LIN {X 0.201,Y -554.749,Z 1469.573,A 0.000,B 0.000,C 90.000,E1 139.013} C_DIS
LIN {X -0.001,Y -555.947,Z 1469.566,A 0.000,B 0.000,C 90.000,E1 137.919} C_DIS
LIN {X -0.117,Y -557.300,Z 1469.559,A 0.000,B 0.000,C 90.000,E1 136.539} C_DIS
LIN {X 0.103,Y -558.249,Z 1469.552,A 0.000,B 0.000,C 90.000,E1 135.405} C_DIS
LIN {X 0.340,Y -559.051,Z 1469.546,A 0.000,B 0.000,C 90.000,E1 134.271} C_DIS
LIN {X 0.127,Y -559.624,Z 1469.542,A 0.000,B 0.000,C 90.000,E1 133.461} C_DIS
LIN {X 0.073,Y -560.260,Z 1469.534,A 0.000,B 0.000,C 90.000,E1 132.081} C_DIS
LIN {X -0.054,Y -560.649,Z 1469.528,A 0.000,B 0.000,C 90.000,E1 130.987} C_DIS
LIN {X -0.119,Y -560.823,Z 1469.522,A 0.000,B 0.000,C 90.000,E1 129.886} C_DIS
LIN {X -0.071,Y -560.958,Z 1469.512,A 0.000,B 0.000,C 90.000,E1 128.222} C_DIS
LIN {X -0.281,Y -561.117,Z 1469.503,A 0.000,B 0.000,C 90.000,E1 126.583} C_DIS
LIN {X 0.009,Y -561.144,Z 1469.499,A 0.000,B 0.000,C 90.000,E1 125.724} C_DIS
LIN {X 0.070,Y -560.901,Z 1469.492,A 0.000,B 0.000,C 90.000,E1 124.612} C_DIS
LIN {X -0.171,Y -560.446,Z 1469.475,A 0.000,B 0.000,C 90.000,E1 121.592} C_DIS
LIN {X 0.273,Y -560.571,Z 1469.463,A 0.000,B 0.000,C 90.000,E1 119.333} C_DIS
LIN {X -0.178,Y -560.837,Z 1469.454,A 0.000,B 0.000,C 90.000,E1 117.719} C_DIS
LIN {X -0.115,Y -561.178,Z 1469.445,A 0.000,B 0.000,C 90.000,E1 116.052} C_DIS
LIN {X 0.259,Y -561.729,Z 1469.434,A 0.000,B 0.000,C 90.000,E1 114.079} C_DIS
LIN {X 0.068,Y -562.198,Z 1469.426,A 0.000,B 0.000,C 90.000,E1 112.717} C_DIS
LIN {X 0.210,Y -562.729,Z 1469.417,A 0.000,B 0.000,C 90.000,E1 111.046} C_DIS
LIN {X -0.057,Y -563.216,Z 1469.406,A 0.000,B 0.000,C 90.000,E1 109.141} C_DIS
LIN {X -0.074,Y -563.557,Z 1469.399,A 0.000,B 0.000,C 90.000,E1 107.764} C_DIS
LIN {X -0.154,Y -564.110,Z 1469.388,A 0.000,B 0.000,C 90.000,E1 105.843} C_DIS
LIN {X 0.159,Y -564.750,Z 1469.377,A 0.000,B 0.000,C 90.000,E1 103.883} C_DIS
LIN {X -0.160,Y -565.614,Z 1469.365,A 0.000,B 0.000,C 90.000,E1 101.715} C_DIS
LIN {X -0.004,Y -566.581,Z 1469.353,A 0.000,B 0.000,C 90.000,E1 99.500} C_DIS
LIN {X -0.090,Y -567.411,Z 1469.342,A 0.000,B 0.000,C 90.000,E1 97.587} C_DIS
LIN {X -0.232,Y -568.473,Z 1469.332,A 0.000,B 0.000,C 90.000,E1 95.682} C_DIS
LIN {X -0.289,Y -569.933,Z 1469.319,A 0.000,B 0.000,C 90.000,E1 93.498} C_DIS
LIN {X 0.091,Y -571.319,Z 1469.309,A 0.000,B 0.000,C 90.000,E1 91.547} C_DIS
LIN {X 0.042,Y -573.033,Z 1469.297,A 0.000,B 0.000,C 90.000,E1 89.370} C_DIS
LIN {X -0.237,Y -574.312,Z 1469.287,A 0.000,B 0.000,C 90.000,E1 87.764} C_DIS
LIN {X 0.267,Y -575.826,Z 1469.277,A 0.000,B 0.000,C 90.000,E1 85.812} C_DIS
LIN {X 0.077,Y -577.153,Z 1469.268,A 0.000,B 0.000,C 90.000,E1 84.204} C_DIS
LIN {X 0.174,Y -578.805,Z 1469.257,A 0.000,B 0.000,C 90.000,E1 82.299} C_DIS
LIN {X -0.181,Y -580.471,Z 1469.247,A 0.000,B 0.000,C 90.000,E1 80.443} C_DIS
LIN {X -0.058,Y -581.907,Z 1469.238,A 0.000,B 0.000,C 90.000,E1 78.814} C_DIS
LIN {X -0.125,Y -583.585,Z 1469.227,A 0.000,B 0.000,C 90.000,E1 76.937} C_DIS
LIN {X 0.019,Y -584.286,Z 1469.223,A 0.000,B 0.000,C 90.000,E1 76.117} C_DIS
LIN {X -0.015,Y -585.019,Z 1469.217,A 0.000,B 0.000,C 90.000,E1 75.046} C_DIS
LIN {X -0.127,Y -585.954,Z 1469.208,A 0.000,B 0.000,C 90.000,E1 73.449} C_DIS
LIN {X 0.114,Y -586.813,Z 1469.199,A 0.000,B 0.000,C 90.000,E1 71.819} C_DIS
LIN {X -0.177,Y -587.738,Z 1469.190,A 0.000,B 0.000,C 90.000,E1 70.242} C_DIS
LIN {X -0.122,Y -588.454,Z 1469.183,A 0.000,B 0.000,C 90.000,E1 68.901} C_DIS
LIN {X 0.129,Y -589.641,Z 1469.171,A 0.000,B 0.000,C 90.000,E1 66.741} C_DIS
LIN {X -0.084,Y -590.787,Z 1469.161,A 0.000,B 0.000,C 90.000,E1 64.897} C_DIS
LIN {X -0.156,Y -591.847,Z 1469.152,A 0.000,B 0.000,C 90.000,E1 63.307} C_DIS
LIN {X -0.334,Y -593.772,Z 1469.137,A 0.000,B 0.000,C 90.000,E1 60.667} C_DIS
LIN {X -0.115,Y -595.362,Z 1469.127,A 0.000,B 0.000,C 90.000,E1 58.791} C_DIS
LIN {X 0.370,Y -597.188,Z 1469.115,A 0.000,B 0.000,C 90.000,E1 56.628} C_DIS
LIN {X 0.022,Y -598.277,Z 1469.108,A 0.000,B 0.000,C 90.000,E1 55.341} C_DIS
LIN {X -0.114,Y -599.280,Z 1469.100,A 0.000,B 0.000,C 90.000,E1 54.036} C_DIS
LIN {X -0.089,Y -600.482,Z 1469.090,A 0.000,B 0.000,C 90.000,E1 52.190} C_DIS
LIN {X -0.177,Y -601.393,Z 1469.083,A 0.000,B 0.000,C 90.000,E1 50.884} C_DIS
LIN {X -0.118,Y -601.869,Z 1469.077,A 0.000,B 0.000,C 90.000,E1 49.828} C_DIS
LIN {X -0.016,Y -602.241,Z 1469.068,A 0.000,B 0.000,C 90.000,E1 48.243} C_DIS
LIN {X 0.047,Y -602.454,Z 1469.062,A 0.000,B 0.000,C 90.000,E1 47.187} C_DIS
LIN {X -0.325,Y -602.466,Z 1469.053,A 0.000,B 0.000,C 90.000,E1 45.648} C_DIS
LIN {X 0.365,Y -601.994,Z 1469.046,A 0.000,B 0.000,C 90.000,E1 44.271} C_DIS
LIN {X -0.249,Y -601.593,Z 1469.042,A 0.000,B 0.000,C 90.000,E1 43.542} C_DIS
LIN {X 0.211,Y -600.855,Z 1469.036,A 0.000,B 0.000,C 90.000,E1 42.447} C_DIS
LIN {X -0.191,Y -599.900,Z 1469.030,A 0.000,B 0.000,C 90.000,E1 41.434} C_DIS
LIN {X -0.157,Y -598.721,Z 1469.024,A 0.000,B 0.000,C 90.000,E1 40.378} C_DIS
LIN {X 0.320,Y -597.355,Z 1469.018,A 0.000,B 0.000,C 90.000,E1 39.277} C_DIS
LIN {X -0.056,Y -595.749,Z 1469.013,A 0.000,B 0.000,C 90.000,E1 38.257} C_DIS
LIN {X 0.157,Y -594.560,Z 1469.008,A 0.000,B 0.000,C 90.000,E1 37.443} C_DIS
LIN {X -0.047,Y -592.134,Z 1469.001,A 0.000,B 0.000,C 90.000,E1 36.137} C_DIS
LIN {X -0.163,Y -589.103,Z 1468.993,A 0.000,B 0.000,C 90.000,E1 34.818} C_DIS
LIN {X 0.295,Y -586.164,Z 1468.987,A 0.000,B 0.000,C 90.000,E1 33.706} C_DIS
LIN {X -0.280,Y -583.793,Z 1468.983,A 0.000,B 0.000,C 90.000,E1 32.959} C_DIS
LIN {X -0.073,Y -581.068,Z 1468.979,A 0.000,B 0.000,C 90.000,E1 32.133} C_DIS
LIN {X -0.203,Y -578.020,Z 1468.974,A 0.000,B 0.000,C 90.000,E1 31.337} C_DIS
LIN {X -0.066,Y -574.598,Z 1468.969,A 0.000,B 0.000,C 90.000,E1 30.512} C_DIS
LIN {X 0.312,Y -571.404,Z 1468.966,A 0.000,B 0.000,C 90.000,E1 29.795} C_DIS
LIN {X 0.075,Y -567.170,Z 1468.961,A 0.000,B 0.000,C 90.000,E1 28.999} C_DIS
LIN {X -0.288,Y -564.172,Z 1468.958,A 0.000,B 0.000,C 90.000,E1 28.487} C_DIS
LIN {X -0.003,Y -560.134,Z 1468.954,A 0.000,B 0.000,C 90.000,E1 27.769} C_DIS
LIN {X -0.016,Y -555.858,Z 1468.950,A 0.000,B 0.000,C 90.000,E1 27.078} C_DIS
LIN {X -0.155,Y -548.245,Z 1468.944,A 0.000,B 0.000,C 90.000,E1 25.976} C_DIS
LIN {X 0.206,Y -540.958,Z 1468.939,A 0.000,B 0.000,C 90.000,E1 24.951} C_DIS
LIN {X 0.029,Y -535.255,Z 1468.935,A 0.000,B 0.000,C 90.000,E1 24.259} C_DIS
LIN {X 0.142,Y -528.093,Z 1468.930,A 0.000,B 0.000,C 90.000,E1 23.387} C_DIS
LIN {X 0.221,Y -523.920,Z 1468.928,A 0.000,B 0.000,C 90.000,E1 22.950} C_DIS
LIN {X -0.100,Y -520.939,Z 1468.926,A 0.000,B 0.000,C 90.000,E1 22.717} C_DIS
LIN {X -0.056,Y -517.716,Z 1468.925,A 0.000,B 0.000,C 90.000,E1 22.461} C_DIS
LIN {X 0.056,Y -516.052,Z 1468.924,A 0.000,B 0.000,C 90.000,E1 22.333} C_DIS
LIN {X 0.011,Y -512.686,Z 1468.923,A 0.000,B 0.000,C 90.000,E1 22.153} C_DIS
LIN {X 0.005,Y -510.601,Z 1468.923,A 0.000,B 0.000,C 90.000,E1 22.078} C_DIS
LIN {X -0.187,Y -509.425,Z 1468.923,A 0.000,B 0.000,C 90.000,E1 22.078} C_DIS
LIN {X 0.188,Y -378.596,Z 1468.923,A 0.000,B 0.000,C 90.000,E1 22.025} C_DIS
LIN {X 0.122,Y -373.766,Z 1468.898,A 0.000,B 0.000,C 90.000,E1 17.638} C_DIS
LIN {X 0.069,Y -372.871,Z 1468.894,A 0.000,B 0.000,C 90.000,E1 16.913} C_DIS
LIN {X -0.029,Y -367.601,Z 1468.865,A 0.000,B 0.000,C 90.000,E1 11.771} C_DIS
LIN {X 0.055,Y -366.481,Z 1468.855,A 0.000,B 0.000,C 90.000,E1 9.905} C_DIS
LIN {X -0.009,Y -361.784,Z 1468.822,A 0.000,B 0.000,C 90.000,E1 3.955} C_DIS
LIN {X -0.123,Y -360.899,Z 1468.801,A 0.000,B 0.000,C 90.000,E1 0.229} C_DIS
LIN {X -0.053,Y -359.426,Z 1468.770,A 0.000,B 0.000,C 90.000,E1 354.546} C_DIS
LIN {X 0.070,Y -358.890,Z 1468.759,A 0.000,B 0.000,C 90.000,E1 352.648} C_DIS
LIN {X -0.020,Y -359.563,Z 1468.726,A 0.000,B 0.000,C 90.000,E1 346.645} C_DIS
LIN {X 0.001,Y -361.801,Z 1468.684,A 0.000,B 0.000,C 90.000,E1 339.135} C_DIS
LIN {X -0.154,Y -362.053,Z 1468.680,A 0.000,B 0.000,C 90.000,E1 338.411} C_DIS
LIN {X 0.189,Y -365.980,Z 1468.643,A 0.000,B 0.000,C 90.000,E1 331.641} C_DIS
LIN {X 0.029,Y -366.387,Z 1468.639,A 0.000,B 0.000,C 90.000,E1 330.923} C_DIS
LIN {X -0.031,Y -371.355,Z 1468.604,A 0.000,B 0.000,C 90.000,E1 324.642} C_DIS
LIN {X -0.043,Y -371.766,Z 1468.602,A 0.000,B 0.000,C 90.000,E1 324.276} C_DIS
LIN {X 0.013,Y -377.358,Z 1468.567,A 0.000,B 0.000,C 90.000,E1 318.038} C_DIS
LIN {X 0.012,Y -378.235,Z 1468.563,A 0.000,B 0.000,C 90.000,E1 317.310} C_DIS
LIN {X 0.002,Y -383.940,Z 1468.531,A 0.000,B 0.000,C 90.000,E1 311.515} C_DIS
LIN {X 0.088,Y -384.893,Z 1468.527,A 0.000,B 0.000,C 90.000,E1 310.782} C_DIS
LIN {X 0.262,Y -390.610,Z 1468.495,A 0.000,B 0.000,C 90.000,E1 305.025} C_DIS
LIN {X 0.106,Y -391.104,Z 1468.493,A 0.000,B 0.000,C 90.000,E1 304.692} C_DIS
LIN {X 0.022,Y -391.648,Z 1468.489,A 0.000,B 0.000,C 90.000,E1 303.992} C_DIS
LIN {X -0.080,Y -396.825,Z 1468.459,A 0.000,B 0.000,C 90.000,E1 298.693} C_DIS
LIN {X -0.210,Y -397.120,Z 1468.457,A 0.000,B 0.000,C 90.000,E1 298.359} C_DIS
LIN {X -0.055,Y -401.597,Z 1468.426,A 0.000,B 0.000,C 90.000,E1 292.717} C_DIS
LIN {X 0.222,Y -404.659,Z 1468.395,A 0.000,B 0.000,C 90.000,E1 287.094} C_DIS
LIN {X -0.079,Y -404.735,Z 1468.391,A 0.000,B 0.000,C 90.000,E1 286.441} C_DIS
LIN {X 0.214,Y -406.099,Z 1468.364,A 0.000,B 0.000,C 90.000,E1 281.535} C_DIS
LIN {X -0.176,Y -406.094,Z 1468.362,A 0.000,B 0.000,C 90.000,E1 281.243} C_DIS
LIN {X -0.097,Y -405.680,Z 1468.333,A 0.000,B 0.000,C 90.000,E1 276.024} C_DIS
LIN {X -0.165,Y -405.058,Z 1468.328,A 0.000,B 0.000,C 90.000,E1 274.992} C_DIS
LIN {X -0.060,Y -403.497,Z 1468.304,A 0.000,B 0.000,C 90.000,E1 270.802} C_DIS
LIN {X -0.092,Y -403.288,Z 1468.302,A 0.000,B 0.000,C 90.000,E1 270.458} C_DIS
LIN {X 0.091,Y -398.931,Z 1468.271,A 0.000,B 0.000,C 90.000,E1 264.837} C_DIS
LIN {X -0.040,Y -393.108,Z 1468.242,A 0.000,B 0.000,C 90.000,E1 259.567} C_DIS
LIN {X -0.079,Y -392.835,Z 1468.240,A 0.000,B 0.000,C 90.000,E1 259.218} C_DIS
LIN {X 0.034,Y -385.993,Z 1468.212,A 0.000,B 0.000,C 90.000,E1 254.212} C_DIS
LIN {X -0.026,Y -385.267,Z 1468.208,A 0.000,B 0.000,C 90.000,E1 253.504} C_DIS
LIN {X -0.004,Y -384.768,Z 1468.206,A 0.000,B 0.000,C 90.000,E1 253.142} C_DIS
LIN {X 0.221,Y -377.973,Z 1468.182,A 0.000,B 0.000,C 90.000,E1 248.773} C_DIS
LIN {X -0.044,Y -376.233,Z 1468.174,A 0.000,B 0.000,C 90.000,E1 247.358} C_DIS
LIN {X 0.057,Y -374.944,Z 1468.170,A 0.000,B 0.000,C 90.000,E1 246.613} C_DIS
LIN {X -0.208,Y -368.417,Z 1468.148,A 0.000,B 0.000,C 90.000,E1 242.615} C_DIS
LIN {X 0.097,Y -366.047,Z 1468.137,A 0.000,B 0.000,C 90.000,E1 240.717} C_DIS
LIN {X 0.004,Y -359.196,Z 1468.115,A 0.000,B 0.000,C 90.000,E1 236.628} C_DIS
LIN {X 0.021,Y -355.842,Z 1468.100,A 0.000,B 0.000,C 90.000,E1 233.989} C_DIS
LIN {X -0.173,Y -348.793,Z 1468.075,A 0.000,B 0.000,C 90.000,E1 229.461} C_DIS
LIN {X -0.097,Y -346.185,Z 1468.062,A 0.000,B 0.000,C 90.000,E1 227.148} C_DIS
LIN {X -0.088,Y -345.065,Z 1468.058,A 0.000,B 0.000,C 90.000,E1 226.377} C_DIS
LIN {X 0.094,Y -338.586,Z 1468.030,A 0.000,B 0.000,C 90.000,E1 221.310} C_DIS
LIN {X 0.094,Y -336.840,Z 1468.019,A 0.000,B 0.000,C 90.000,E1 219.358} C_DIS
LIN {X 0.014,Y -330.861,Z 1467.988,A 0.000,B 0.000,C 90.000,E1 213.865} C_DIS
LIN {X 0.149,Y -329.296,Z 1467.975,A 0.000,B 0.000,C 90.000,E1 211.465} C_DIS
LIN {X -0.154,Y -324.669,Z 1467.942,A 0.000,B 0.000,C 90.000,E1 205.540} C_DIS
LIN {X 0.174,Y -323.837,Z 1467.928,A 0.000,B 0.000,C 90.000,E1 203.078} C_DIS
LIN {X -0.017,Y -321.124,Z 1467.881,A 0.000,B 0.000,C 90.000,E1 194.662} C_DIS
LIN {X 0.138,Y -320.932,Z 1467.877,A 0.000,B 0.000,C 90.000,E1 193.828} C_DIS
LIN {X -0.076,Y -321.562,Z 1467.832,A 0.000,B 0.000,C 90.000,E1 185.796} C_DIS
LIN {X -0.143,Y -324.415,Z 1467.790,A 0.000,B 0.000,C 90.000,E1 178.165} C_DIS
LIN {X -0.141,Y -325.376,Z 1467.783,A 0.000,B 0.000,C 90.000,E1 176.963} C_DIS
LIN {X -0.100,Y -329.112,Z 1467.750,A 0.000,B 0.000,C 90.000,E1 170.971} C_DIS
LIN {X 0.061,Y -334.260,Z 1467.726,A 0.000,B 0.000,C 90.000,E1 166.589} C_DIS
LIN {X 0.067,Y -335.488,Z 1467.719,A 0.000,B 0.000,C 90.000,E1 165.408} C_DIS
LIN {X 0.143,Y -340.932,Z 1467.695,A 0.000,B 0.000,C 90.000,E1 161.094} C_DIS
LIN {X -0.172,Y -342.138,Z 1467.691,A 0.000,B 0.000,C 90.000,E1 160.369} C_DIS
LIN {X 0.102,Y -347.570,Z 1467.668,A 0.000,B 0.000,C 90.000,E1 156.305} C_DIS
LIN {X 0.097,Y -466.149,Z 1467.668,A 0.000,B 0.000,C 90.000,E1 156.305} C_DIS
LIN {X 0.196,Y -469.174,Z 1467.668,A 0.000,B 0.000,C 90.000,E1 156.230} C_DIS
LIN {X -0.079,Y -473.073,Z 1467.667,A 0.000,B 0.000,C 90.000,E1 156.102} C_DIS
LIN {X 0.134,Y -475.940,Z 1467.666,A 0.000,B 0.000,C 90.000,E1 155.921} C_DIS
LIN {X 0.123,Y -478.786,Z 1467.665,A 0.000,B 0.000,C 90.000,E1 155.741} C_DIS
LIN {X 0.219,Y -483.218,Z 1467.664,A 0.000,B 0.000,C 90.000,E1 155.409} C_DIS
LIN {X -0.194,Y -488.987,Z 1467.661,A 0.000,B 0.000,C 90.000,E1 154.973} C_DIS
LIN {X -0.117,Y -497.335,Z 1467.656,A 0.000,B 0.000,C 90.000,E1 154.152} C_DIS
LIN {X 0.163,Y -500.136,Z 1467.655,A 0.000,B 0.000,C 90.000,E1 153.845} C_DIS
LIN {X -0.135,Y -505.377,Z 1467.652,A 0.000,B 0.000,C 90.000,E1 153.307} C_DIS
LIN {X 0.082,Y -510.366,Z 1467.648,A 0.000,B 0.000,C 90.000,E1 152.692} C_DIS
LIN {X 0.062,Y -514.904,Z 1467.645,A 0.000,B 0.000,C 90.000,E1 152.103} C_DIS
LIN {X 0.071,Y -518.945,Z 1467.642,A 0.000,B 0.000,C 90.000,E1 151.513} C_DIS
LIN {X 0.111,Y -522.546,Z 1467.639,A 0.000,B 0.000,C 90.000,E1 150.923} C_DIS
LIN {X 0.179,Y -525.767,Z 1467.635,A 0.000,B 0.000,C 90.000,E1 150.333} C_DIS
LIN {X 0.115,Y -529.332,Z 1467.631,A 0.000,B 0.000,C 90.000,E1 149.616} C_DIS
LIN {X -0.227,Y -531.880,Z 1467.628,A 0.000,B 0.000,C 90.000,E1 149.076} C_DIS
LIN {X 0.181,Y -534.218,Z 1467.625,A 0.000,B 0.000,C 90.000,E1 148.456} C_DIS
LIN {X 0.321,Y -537.331,Z 1467.620,A 0.000,B 0.000,C 90.000,E1 147.582} C_DIS
LIN {X 0.041,Y -540.071,Z 1467.615,A 0.000,B 0.000,C 90.000,E1 146.755} C_DIS
LIN {X 0.240,Y -542.557,Z 1467.611,A 0.000,B 0.000,C 90.000,E1 145.881} C_DIS
LIN {X 0.010,Y -544.834,Z 1467.606,A 0.000,B 0.000,C 90.000,E1 145.055} C_DIS
LIN {X 0.160,Y -547.458,Z 1467.600,A 0.000,B 0.000,C 90.000,E1 143.909} C_DIS
LIN {X 0.022,Y -549.701,Z 1467.593,A 0.000,B 0.000,C 90.000,E1 142.798} C_DIS
LIN {X -0.253,Y -551.173,Z 1467.589,A 0.000,B 0.000,C 90.000,E1 141.984} C_DIS
LIN {X 0.330,Y -552.833,Z 1467.583,A 0.000,B 0.000,C 90.000,E1 140.803} C_DIS
LIN {X 0.159,Y -554.204,Z 1467.576,A 0.000,B 0.000,C 90.000,E1 139.703} C_DIS
LIN {X 0.010,Y -555.758,Z 1467.568,A 0.000,B 0.000,C 90.000,E1 138.324} C_DIS
LIN {X -0.072,Y -557.378,Z 1467.559,A 0.000,B 0.000,C 90.000,E1 136.662} C_DIS
LIN {X -0.235,Y -558.335,Z 1467.553,A 0.000,B 0.000,C 90.000,E1 135.567} C_DIS
LIN {X 0.003,Y -559.169,Z 1467.547,A 0.000,B 0.000,C 90.000,E1 134.433} C_DIS
LIN {X -0.085,Y -559.968,Z 1467.539,A 0.000,B 0.000,C 90.000,E1 133.056} C_DIS
LIN {X -0.136,Y -560.558,Z 1467.531,A 0.000,B 0.000,C 90.000,E1 131.676} C_DIS
LIN {X -0.177,Y -560.849,Z 1467.524,A 0.000,B 0.000,C 90.000,E1 130.297} C_DIS
LIN {X -0.146,Y -560.969,Z 1467.516,A 0.000,B 0.000,C 90.000,E1 128.910} C_DIS
LIN {X 0.091,Y -561.146,Z 1467.505,A 0.000,B 0.000,C 90.000,E1 126.950} C_DIS
LIN {X 0.027,Y -561.184,Z 1467.499,A 0.000,B 0.000,C 90.000,E1 125.851} C_DIS
LIN {X -0.012,Y -561.036,Z 1467.495,A 0.000,B 0.000,C 90.000,E1 125.025} C_DIS
LIN {X -0.033,Y -560.452,Z 1467.479,A 0.000,B 0.000,C 90.000,E1 122.260} C_DIS
LIN {X -0.151,Y -560.474,Z 1467.469,A 0.000,B 0.000,C 90.000,E1 120.335} C_DIS
LIN {X 0.024,Y -560.750,Z 1467.456,A 0.000,B 0.000,C 90.000,E1 118.103} C_DIS
LIN {X 0.082,Y -561.087,Z 1467.447,A 0.000,B 0.000,C 90.000,E1 116.437} C_DIS
LIN {X 0.259,Y -561.706,Z 1467.435,A 0.000,B 0.000,C 90.000,E1 114.207} C_DIS
LIN {X -0.132,Y -562.266,Z 1467.425,A 0.000,B 0.000,C 90.000,E1 112.589} C_DIS
LIN {X 0.008,Y -562.769,Z 1467.416,A 0.000,B 0.000,C 90.000,E1 110.918} C_DIS
LIN {X 0.270,Y -563.294,Z 1467.406,A 0.000,B 0.000,C 90.000,E1 108.960} C_DIS
LIN {X -0.205,Y -563.516,Z 1467.401,A 0.000,B 0.000,C 90.000,E1 108.181} C_DIS
LIN {X -0.289,Y -564.022,Z 1467.390,A 0.000,B 0.000,C 90.000,E1 106.260} C_DIS
LIN {X 0.187,Y -564.730,Z 1467.378,A 0.000,B 0.000,C 90.000,E1 104.008} C_DIS
LIN {X -0.005,Y -565.596,Z 1467.366,A 0.000,B 0.000,C 90.000,E1 101.827} C_DIS
LIN {X -0.029,Y -566.416,Z 1467.355,A 0.000,B 0.000,C 90.000,E1 99.905} C_DIS
LIN {X 0.181,Y -567.017,Z 1467.347,A 0.000,B 0.000,C 90.000,E1 98.511} C_DIS
LIN {X -0.264,Y -568.258,Z 1467.334,A 0.000,B 0.000,C 90.000,E1 96.087} C_DIS
LIN {X -0.159,Y -569.888,Z 1467.320,A 0.000,B 0.000,C 90.000,E1 93.612} C_DIS
LIN {X 0.220,Y -571.259,Z 1467.309,A 0.000,B 0.000,C 90.000,E1 91.661} C_DIS
LIN {X -0.111,Y -572.525,Z 1467.300,A 0.000,B 0.000,C 90.000,E1 90.057} C_DIS
LIN {X 0.018,Y -573.646,Z 1467.293,A 0.000,B 0.000,C 90.000,E1 88.682} C_DIS
LIN {X -0.252,Y -574.959,Z 1467.284,A 0.000,B 0.000,C 90.000,E1 87.078} C_DIS
LIN {X 0.110,Y -576.250,Z 1467.275,A 0.000,B 0.000,C 90.000,E1 85.412} C_DIS
LIN {X -0.224,Y -577.403,Z 1467.267,A 0.000,B 0.000,C 90.000,E1 84.090} C_DIS
LIN {X -0.125,Y -579.057,Z 1467.257,A 0.000,B 0.000,C 90.000,E1 82.186} C_DIS
LIN {X 0.092,Y -580.736,Z 1467.246,A 0.000,B 0.000,C 90.000,E1 80.274} C_DIS
LIN {X 0.327,Y -582.230,Z 1467.237,A 0.000,B 0.000,C 90.000,E1 78.634} C_DIS
LIN {X -0.053,Y -584.147,Z 1467.225,A 0.000,B 0.000,C 90.000,E1 76.520} C_DIS
LIN {X 0.098,Y -584.759,Z 1467.221,A 0.000,B 0.000,C 90.000,E1 75.700} C_DIS
LIN {X 0.073,Y -585.441,Z 1467.215,A 0.000,B 0.000,C 90.000,E1 74.629} C_DIS
LIN {X 0.138,Y -586.351,Z 1467.206,A 0.000,B 0.000,C 90.000,E1 73.015} C_DIS
LIN {X 0.214,Y -587.207,Z 1467.197,A 0.000,B 0.000,C 90.000,E1 71.402} C_DIS
LIN {X 0.258,Y -588.014,Z 1467.189,A 0.000,B 0.000,C 90.000,E1 70.061} C_DIS
LIN {X 0.194,Y -588.824,Z 1467.181,A 0.000,B 0.000,C 90.000,E1 68.465} C_DIS
LIN {X 0.141,Y -589.732,Z 1467.172,A 0.000,B 0.000,C 90.000,E1 66.869} C_DIS
LIN {X -0.074,Y -590.881,Z 1467.161,A 0.000,B 0.000,C 90.000,E1 65.025} C_DIS
LIN {X 0.284,Y -592.149,Z 1467.151,A 0.000,B 0.000,C 90.000,E1 63.127} C_DIS
LIN {X -0.121,Y -594.089,Z 1467.136,A 0.000,B 0.000,C 90.000,E1 60.511} C_DIS
LIN {X -0.189,Y -595.677,Z 1467.126,A 0.000,B 0.000,C 90.000,E1 58.663} C_DIS
LIN {X 0.074,Y -597.286,Z 1467.116,A 0.000,B 0.000,C 90.000,E1 56.786} C_DIS
LIN {X 0.295,Y -598.634,Z 1467.107,A 0.000,B 0.000,C 90.000,E1 55.182} C_DIS
LIN {X -0.182,Y -599.616,Z 1467.099,A 0.000,B 0.000,C 90.000,E1 53.909} C_DIS
LIN {X -0.157,Y -600.796,Z 1467.089,A 0.000,B 0.000,C 90.000,E1 52.065} C_DIS
LIN {X -0.113,Y -601.577,Z 1467.083,A 0.000,B 0.000,C 90.000,E1 51.009} C_DIS
LIN {X -0.046,Y -602.091,Z 1467.078,A 0.000,B 0.000,C 90.000,E1 49.952} C_DIS
LIN {X 0.313,Y -602.538,Z 1467.067,A 0.000,B 0.000,C 90.000,E1 48.081} C_DIS
LIN {X -0.061,Y -602.725,Z 1467.062,A 0.000,B 0.000,C 90.000,E1 47.067} C_DIS
LIN {X 0.217,Y -602.743,Z 1467.054,A 0.000,B 0.000,C 90.000,E1 45.729} C_DIS
LIN {X 0.039,Y -602.531,Z 1467.050,A 0.000,B 0.000,C 90.000,E1 44.960} C_DIS
LIN {X 0.302,Y -601.979,Z 1467.043,A 0.000,B 0.000,C 90.000,E1 43.623} C_DIS
LIN {X 0.125,Y -601.440,Z 1467.038,A 0.000,B 0.000,C 90.000,E1 42.852} C_DIS
LIN {X -0.028,Y -600.376,Z 1467.031,A 0.000,B 0.000,C 90.000,E1 41.553} C_DIS
LIN {X -0.198,Y -598.867,Z 1467.024,A 0.000,B 0.000,C 90.000,E1 40.253} C_DIS
LIN {X -0.175,Y -597.455,Z 1467.018,A 0.000,B 0.000,C 90.000,E1 39.197} C_DIS
LIN {X -0.092,Y -595.069,Z 1467.009,A 0.000,B 0.000,C 90.000,E1 37.604} C_DIS
LIN {X -0.113,Y -594.169,Z 1467.006,A 0.000,B 0.000,C 90.000,E1 37.076} C_DIS
LIN {X -0.061,Y -592.208,Z 1467.000,A 0.000,B 0.000,C 90.000,E1 36.011} C_DIS
LIN {X -0.172,Y -589.101,Z 1466.993,A 0.000,B 0.000,C 90.000,E1 34.692} C_DIS
LIN {X -0.333,Y -585.389,Z 1466.985,A 0.000,B 0.000,C 90.000,E1 33.372} C_DIS
LIN {X 0.033,Y -583.794,Z 1466.982,A 0.000,B 0.000,C 90.000,E1 32.801} C_DIS
LIN {X -0.074,Y -581.018,Z 1466.978,A 0.000,B 0.000,C 90.000,E1 32.005} C_DIS
LIN {X -0.202,Y -577.937,Z 1466.973,A 0.000,B 0.000,C 90.000,E1 31.209} C_DIS
LIN {X -0.066,Y -574.532,Z 1466.969,A 0.000,B 0.000,C 90.000,E1 30.384} C_DIS
LIN {X 0.312,Y -571.272,Z 1466.965,A 0.000,B 0.000,C 90.000,E1 29.667} C_DIS
LIN {X 0.075,Y -567.034,Z 1466.960,A 0.000,B 0.000,C 90.000,E1 28.871} C_DIS
LIN {X 0.286,Y -562.409,Z 1466.956,A 0.000,B 0.000,C 90.000,E1 28.025} C_DIS
LIN {X 0.086,Y -556.524,Z 1466.951,A 0.000,B 0.000,C 90.000,E1 27.078} C_DIS
LIN {X -0.046,Y -548.994,Z 1466.944,A 0.000,B 0.000,C 90.000,E1 25.976} C_DIS
LIN {X -0.033,Y -540.645,Z 1466.938,A 0.000,B 0.000,C 90.000,E1 24.847} C_DIS
LIN {X 0.153,Y -536.107,Z 1466.935,A 0.000,B 0.000,C 90.000,E1 24.259} C_DIS
LIN {X 0.123,Y -527.736,Z 1466.929,A 0.000,B 0.000,C 90.000,E1 23.259} C_DIS
LIN {X 0.004,Y -522.522,Z 1466.926,A 0.000,B 0.000,C 90.000,E1 22.695} C_DIS
LIN {X 0.003,Y -518.208,Z 1466.924,A 0.000,B 0.000,C 90.000,E1 22.280} C_DIS
LIN {X -0.007,Y -513.505,Z 1466.922,A 0.000,B 0.000,C 90.000,E1 21.897} C_DIS
LIN {X 0.047,Y -511.740,Z 1466.921,A 0.000,B 0.000,C 90.000,E1 21.770} C_DIS
LIN {X 0.031,Y -509.876,Z 1466.920,A 0.000,B 0.000,C 90.000,E1 21.663} C_DIS
LIN {X -0.001,Y -506.943,Z 1466.920,A 0.000,B 0.000,C 90.000,E1 21.535} C_DIS
LIN {X 0.199,Y -504.735,Z 1466.919,A 0.000,B 0.000,C 90.000,E1 21.461} C_DIS
LIN {X 0.124,Y -377.830,Z 1466.919,A 0.000,B 0.000,C 90.000,E1 21.461} C_DIS
LIN {X -0.114,Y -373.501,Z 1466.897,A 0.000,B 0.000,C 90.000,E1 17.402} C_DIS
LIN {X -0.075,Y -367.945,Z 1466.868,A 0.000,B 0.000,C 90.000,E1 12.243} C_DIS
LIN {X -0.056,Y -366.530,Z 1466.856,A 0.000,B 0.000,C 90.000,E1 10.018} C_DIS
LIN {X 0.087,Y -365.038,Z 1466.847,A 0.000,B 0.000,C 90.000,E1 8.511} C_DIS
LIN {X 0.182,Y -361.084,Z 1466.810,A 0.000,B 0.000,C 90.000,E1 1.776} C_DIS
LIN {X 0.123,Y -360.905,Z 1466.802,A 0.000,B 0.000,C 90.000,E1 0.286} C_DIS
LIN {X -0.053,Y -359.426,Z 1466.770,A 0.000,B 0.000,C 90.000,E1 354.546} C_DIS
LIN {X 0.070,Y -358.890,Z 1466.759,A 0.000,B 0.000,C 90.000,E1 352.648} C_DIS
LIN {X -0.020,Y -359.563,Z 1466.726,A 0.000,B 0.000,C 90.000,E1 346.645} C_DIS
LIN {X 0.001,Y -361.801,Z 1466.684,A 0.000,B 0.000,C 90.000,E1 339.135} C_DIS
LIN {X -0.154,Y -362.053,Z 1466.680,A 0.000,B 0.000,C 90.000,E1 338.411} C_DIS
LIN {X 0.189,Y -365.980,Z 1466.643,A 0.000,B 0.000,C 90.000,E1 331.641} C_DIS
LIN {X 0.029,Y -366.387,Z 1466.639,A 0.000,B 0.000,C 90.000,E1 330.923} C_DIS
LIN {X -0.031,Y -371.355,Z 1466.604,A 0.000,B 0.000,C 90.000,E1 324.642} C_DIS
LIN {X -0.043,Y -371.766,Z 1466.602,A 0.000,B 0.000,C 90.000,E1 324.276} C_DIS
LIN {X 0.013,Y -377.358,Z 1466.567,A 0.000,B 0.000,C 90.000,E1 318.038} C_DIS
LIN {X 0.012,Y -378.235,Z 1466.563,A 0.000,B 0.000,C 90.000,E1 317.310} C_DIS
LIN {X 0.002,Y -383.940,Z 1466.531,A 0.000,B 0.000,C 90.000,E1 311.515} C_DIS
LIN {X 0.088,Y -384.893,Z 1466.527,A 0.000,B 0.000,C 90.000,E1 310.782} C_DIS
LIN {X 0.262,Y -390.610,Z 1466.495,A 0.000,B 0.000,C 90.000,E1 305.025} C_DIS
LIN {X 0.106,Y -391.104,Z 1466.493,A 0.000,B 0.000,C 90.000,E1 304.692} C_DIS
LIN {X 0.022,Y -391.648,Z 1466.489,A 0.000,B 0.000,C 90.000,E1 303.992} C_DIS
LIN {X -0.080,Y -396.825,Z 1466.459,A 0.000,B 0.000,C 90.000,E1 298.693} C_DIS
LIN {X -0.210,Y -397.120,Z 1466.457,A 0.000,B 0.000,C 90.000,E1 298.359} C_DIS
LIN {X -0.055,Y -401.597,Z 1466.426,A 0.000,B 0.000,C 90.000,E1 292.717} C_DIS
LIN {X 0.222,Y -404.659,Z 1466.395,A 0.000,B 0.000,C 90.000,E1 287.094} C_DIS
LIN {X -0.079,Y -404.735,Z 1466.391,A 0.000,B 0.000,C 90.000,E1 286.441} C_DIS
LIN {X 0.214,Y -406.099,Z 1466.364,A 0.000,B 0.000,C 90.000,E1 281.535} C_DIS
LIN {X -0.176,Y -406.094,Z 1466.362,A 0.000,B 0.000,C 90.000,E1 281.243} C_DIS
LIN {X -0.097,Y -405.680,Z 1466.333,A 0.000,B 0.000,C 90.000,E1 276.024} C_DIS
LIN {X -0.165,Y -405.058,Z 1466.328,A 0.000,B 0.000,C 90.000,E1 274.992} C_DIS
LIN {X -0.060,Y -403.497,Z 1466.304,A 0.000,B 0.000,C 90.000,E1 270.802} C_DIS
LIN {X -0.092,Y -403.288,Z 1466.302,A 0.000,B 0.000,C 90.000,E1 270.458} C_DIS
LIN {X 0.091,Y -398.931,Z 1466.271,A 0.000,B 0.000,C 90.000,E1 264.837} C_DIS
LIN {X -0.040,Y -393.108,Z 1466.242,A 0.000,B 0.000,C 90.000,E1 259.567} C_DIS
LIN {X -0.079,Y -392.835,Z 1466.240,A 0.000,B 0.000,C 90.000,E1 259.218} C_DIS
LIN {X 0.034,Y -385.993,Z 1466.212,A 0.000,B 0.000,C 90.000,E1 254.212} C_DIS
LIN {X -0.026,Y -385.267,Z 1466.208,A 0.000,B 0.000,C 90.000,E1 253.504} C_DIS
LIN {X -0.004,Y -384.768,Z 1466.206,A 0.000,B 0.000,C 90.000,E1 253.142} C_DIS
LIN {X 0.221,Y -377.973,Z 1466.182,A 0.000,B 0.000,C 90.000,E1 248.773} C_DIS
LIN {X -0.044,Y -376.233,Z 1466.174,A 0.000,B 0.000,C 90.000,E1 247.358} C_DIS
LIN {X 0.057,Y -374.944,Z 1466.170,A 0.000,B 0.000,C 90.000,E1 246.613} C_DIS
LIN {X -0.208,Y -368.417,Z 1466.148,A 0.000,B 0.000,C 90.000,E1 242.615} C_DIS
LIN {X 0.097,Y -366.047,Z 1466.137,A 0.000,B 0.000,C 90.000,E1 240.717} C_DIS
LIN {X 0.004,Y -359.196,Z 1466.115,A 0.000,B 0.000,C 90.000,E1 236.628} C_DIS
LIN {X 0.021,Y -355.842,Z 1466.100,A 0.000,B 0.000,C 90.000,E1 233.989} C_DIS
LIN {X -0.173,Y -348.793,Z 1466.075,A 0.000,B 0.000,C 90.000,E1 229.461} C_DIS
LIN {X -0.097,Y -346.185,Z 1466.062,A 0.000,B 0.000,C 90.000,E1 227.148} C_DIS
LIN {X -0.088,Y -345.065,Z 1466.058,A 0.000,B 0.000,C 90.000,E1 226.377} C_DIS
LIN {X 0.094,Y -338.586,Z 1466.030,A 0.000,B 0.000,C 90.000,E1 221.310} C_DIS
LIN {X 0.094,Y -336.840,Z 1466.019,A 0.000,B 0.000,C 90.000,E1 219.358} C_DIS
LIN {X 0.014,Y -330.861,Z 1465.988,A 0.000,B 0.000,C 90.000,E1 213.865} C_DIS
LIN {X 0.149,Y -329.296,Z 1465.975,A 0.000,B 0.000,C 90.000,E1 211.465} C_DIS
LIN {X -0.154,Y -324.669,Z 1465.942,A 0.000,B 0.000,C 90.000,E1 205.540} C_DIS
LIN {X 0.174,Y -323.837,Z 1465.928,A 0.000,B 0.000,C 90.000,E1 203.078} C_DIS
LIN {X -0.017,Y -321.124,Z 1465.881,A 0.000,B 0.000,C 90.000,E1 194.662} C_DIS
LIN {X 0.138,Y -320.932,Z 1465.877,A 0.000,B 0.000,C 90.000,E1 193.828} C_DIS
LIN {X -0.076,Y -321.562,Z 1465.832,A 0.000,B 0.000,C 90.000,E1 185.796} C_DIS
LIN {X -0.143,Y -324.415,Z 1465.790,A 0.000,B 0.000,C 90.000,E1 178.165} C_DIS
LIN {X -0.141,Y -325.376,Z 1465.783,A 0.000,B 0.000,C 90.000,E1 176.963} C_DIS
LIN {X -0.100,Y -329.112,Z 1465.750,A 0.000,B 0.000,C 90.000,E1 170.971} C_DIS
LIN {X 0.061,Y -334.260,Z 1465.726,A 0.000,B 0.000,C 90.000,E1 166.589} C_DIS
LIN {X 0.067,Y -335.488,Z 1465.719,A 0.000,B 0.000,C 90.000,E1 165.408} C_DIS
LIN {X 0.143,Y -340.932,Z 1465.695,A 0.000,B 0.000,C 90.000,E1 161.094} C_DIS
LIN {X -0.172,Y -342.138,Z 1465.691,A 0.000,B 0.000,C 90.000,E1 160.369} C_DIS
LIN {X 0.043,Y -346.707,Z 1465.672,A 0.000,B 0.000,C 90.000,E1 156.869} C_DIS
LIN {X 0.018,Y -460.252,Z 1465.672,A 0.000,B 0.000,C 90.000,E1 156.869} C_DIS
LIN {X 0.126,Y -463.257,Z 1465.671,A 0.000,B 0.000,C 90.000,E1 156.794} C_DIS
LIN {X -0.145,Y -465.604,Z 1465.671,A 0.000,B 0.000,C 90.000,E1 156.741} C_DIS
LIN {X -0.158,Y -468.354,Z 1465.670,A 0.000,B 0.000,C 90.000,E1 156.613} C_DIS
LIN {X -0.010,Y -471.281,Z 1465.669,A 0.000,B 0.000,C 90.000,E1 156.433} C_DIS
LIN {X 0.134,Y -474.187,Z 1465.668,A 0.000,B 0.000,C 90.000,E1 156.230} C_DIS
LIN {X 0.024,Y -478.628,Z 1465.666,A 0.000,B 0.000,C 90.000,E1 155.921} C_DIS
LIN {X 0.209,Y -484.407,Z 1465.664,A 0.000,B 0.000,C 90.000,E1 155.409} C_DIS
LIN {X -0.158,Y -491.532,Z 1465.660,A 0.000,B 0.000,C 90.000,E1 154.793} C_DIS
LIN {X 0.116,Y -498.552,Z 1465.656,A 0.000,B 0.000,C 90.000,E1 154.076} C_DIS
LIN {X 0.278,Y -502.524,Z 1465.654,A 0.000,B 0.000,C 90.000,E1 153.640} C_DIS
LIN {X -0.164,Y -506.438,Z 1465.651,A 0.000,B 0.000,C 90.000,E1 153.256} C_DIS
LIN {X -0.001,Y -510.230,Z 1465.649,A 0.000,B 0.000,C 90.000,E1 152.794} C_DIS
LIN {X -0.265,Y -514.804,Z 1465.646,A 0.000,B 0.000,C 90.000,E1 152.231} C_DIS
LIN {X -0.258,Y -518.895,Z 1465.642,A 0.000,B 0.000,C 90.000,E1 151.641} C_DIS
LIN {X -0.220,Y -522.519,Z 1465.639,A 0.000,B 0.000,C 90.000,E1 151.051} C_DIS
LIN {X -0.312,Y -526.527,Z 1465.635,A 0.000,B 0.000,C 90.000,E1 150.333} C_DIS
LIN {X -0.105,Y -530.012,Z 1465.631,A 0.000,B 0.000,C 90.000,E1 149.587} C_DIS
LIN {X 0.018,Y -532.561,Z 1465.628,A 0.000,B 0.000,C 90.000,E1 148.997} C_DIS
LIN {X 0.141,Y -535.895,Z 1465.623,A 0.000,B 0.000,C 90.000,E1 148.122} C_DIS
LIN {X -0.152,Y -536.964,Z 1465.621,A 0.000,B 0.000,C 90.000,E1 147.867} C_DIS
LIN {X 0.010,Y -539.746,Z 1465.617,A 0.000,B 0.000,C 90.000,E1 146.993} C_DIS
LIN {X 0.051,Y -542.259,Z 1465.612,A 0.000,B 0.000,C 90.000,E1 146.135} C_DIS
LIN {X -0.177,Y -544.595,Z 1465.607,A 0.000,B 0.000,C 90.000,E1 145.308} C_DIS
LIN {X 0.099,Y -547.285,Z 1465.601,A 0.000,B 0.000,C 90.000,E1 144.149} C_DIS
LIN {X -0.156,Y -549.596,Z 1465.595,A 0.000,B 0.000,C 90.000,E1 143.050} C_DIS
LIN {X 0.008,Y -551.092,Z 1465.590,A 0.000,B 0.000,C 90.000,E1 142.190} C_DIS
LIN {X 0.186,Y -552.387,Z 1465.585,A 0.000,B 0.000,C 90.000,E1 141.331} C_DIS
LIN {X 0.007,Y -553.870,Z 1465.579,A 0.000,B 0.000,C 90.000,E1 140.231} C_DIS
LIN {X -0.150,Y -555.425,Z 1465.571,A 0.000,B 0.000,C 90.000,E1 138.852} C_DIS
LIN {X 0.072,Y -556.545,Z 1465.565,A 0.000,B 0.000,C 90.000,E1 137.715} C_DIS
LIN {X -0.062,Y -557.861,Z 1465.557,A 0.000,B 0.000,C 90.000,E1 136.338} C_DIS
LIN {X 0.237,Y -558.949,Z 1465.550,A 0.000,B 0.000,C 90.000,E1 134.919} C_DIS
LIN {X 0.026,Y -559.501,Z 1465.545,A 0.000,B 0.000,C 90.000,E1 134.109} C_DIS
LIN {X 0.351,Y -560.262,Z 1465.537,A 0.000,B 0.000,C 90.000,E1 132.690} C_DIS
LIN {X 0.225,Y -560.639,Z 1465.531,A 0.000,B 0.000,C 90.000,E1 131.595} C_DIS
LIN {X -0.179,Y -560.924,Z 1465.524,A 0.000,B 0.000,C 90.000,E1 130.253} C_DIS
LIN {X 0.216,Y -561.017,Z 1465.516,A 0.000,B 0.000,C 90.000,E1 128.830} C_DIS
LIN {X 0.002,Y -561.198,Z 1465.505,A 0.000,B 0.000,C 90.000,E1 126.916} C_DIS
LIN {X 0.056,Y -561.200,Z 1465.499,A 0.000,B 0.000,C 90.000,E1 125.804} C_DIS
LIN {X 0.022,Y -561.046,Z 1465.494,A 0.000,B 0.000,C 90.000,E1 124.978} C_DIS
LIN {X -0.112,Y -560.454,Z 1465.476,A 0.000,B 0.000,C 90.000,E1 121.671} C_DIS
LIN {X -0.221,Y -560.486,Z 1465.465,A 0.000,B 0.000,C 90.000,E1 119.745} C_DIS
LIN {X 0.154,Y -560.771,Z 1465.454,A 0.000,B 0.000,C 90.000,E1 117.769} C_DIS
LIN {X -0.094,Y -561.095,Z 1465.447,A 0.000,B 0.000,C 90.000,E1 116.411} C_DIS
LIN {X -0.168,Y -561.729,Z 1465.434,A 0.000,B 0.000,C 90.000,E1 114.207} C_DIS
LIN {X 0.177,Y -562.302,Z 1465.425,A 0.000,B 0.000,C 90.000,E1 112.514} C_DIS
LIN {X 0.108,Y -562.829,Z 1465.416,A 0.000,B 0.000,C 90.000,E1 110.865} C_DIS
LIN {X -0.235,Y -563.550,Z 1465.402,A 0.000,B 0.000,C 90.000,E1 108.417} C_DIS
LIN {X -0.171,Y -564.065,Z 1465.390,A 0.000,B 0.000,C 90.000,E1 106.205} C_DIS
LIN {X 0.149,Y -564.687,Z 1465.379,A 0.000,B 0.000,C 90.000,E1 104.245} C_DIS
LIN {X -0.043,Y -565.567,Z 1465.367,A 0.000,B 0.000,C 90.000,E1 102.063} C_DIS
LIN {X -0.134,Y -566.257,Z 1465.358,A 0.000,B 0.000,C 90.000,E1 100.423} C_DIS
LIN {X 0.065,Y -566.864,Z 1465.350,A 0.000,B 0.000,C 90.000,E1 99.029} C_DIS
LIN {X -0.197,Y -567.546,Z 1465.341,A 0.000,B 0.000,C 90.000,E1 97.409} C_DIS
LIN {X 0.162,Y -568.638,Z 1465.330,A 0.000,B 0.000,C 90.000,E1 95.454} C_DIS
LIN {X 0.117,Y -570.152,Z 1465.318,A 0.000,B 0.000,C 90.000,E1 93.269} C_DIS
LIN {X -0.064,Y -571.538,Z 1465.308,A 0.000,B 0.000,C 90.000,E1 91.375} C_DIS
LIN {X -0.247,Y -573.099,Z 1465.297,A 0.000,B 0.000,C 90.000,E1 89.484} C_DIS
LIN {X 0.050,Y -574.417,Z 1465.288,A 0.000,B 0.000,C 90.000,E1 87.822} C_DIS
LIN {X 0.229,Y -575.496,Z 1465.280,A 0.000,B 0.000,C 90.000,E1 86.445} C_DIS
LIN {X 0.174,Y -577.097,Z 1465.270,A 0.000,B 0.000,C 90.000,E1 84.552} C_DIS
LIN {X 0.264,Y -578.726,Z 1465.259,A 0.000,B 0.000,C 90.000,E1 82.648} C_DIS
LIN {X 0.255,Y -580.178,Z 1465.250,A 0.000,B 0.000,C 90.000,E1 81.027} C_DIS
LIN {X 0.141,Y -581.379,Z 1465.243,A 0.000,B 0.000,C 90.000,E1 79.690} C_DIS
LIN {X 0.160,Y -582.651,Z 1465.235,A 0.000,B 0.000,C 90.000,E1 78.342} C_DIS
LIN {X 0.118,Y -584.337,Z 1465.225,A 0.000,B 0.000,C 90.000,E1 76.464} C_DIS
LIN {X -0.298,Y -584.959,Z 1465.220,A 0.000,B 0.000,C 90.000,E1 75.700} C_DIS
LIN {X 0.244,Y -585.627,Z 1465.214,A 0.000,B 0.000,C 90.000,E1 74.574} C_DIS
LIN {X 0.308,Y -586.558,Z 1465.206,A 0.000,B 0.000,C 90.000,E1 72.960} C_DIS
LIN {X -0.173,Y -587.403,Z 1465.197,A 0.000,B 0.000,C 90.000,E1 71.402} C_DIS
LIN {X -0.126,Y -588.200,Z 1465.189,A 0.000,B 0.000,C 90.000,E1 70.061} C_DIS
LIN {X 0.243,Y -589.169,Z 1465.179,A 0.000,B 0.000,C 90.000,E1 68.156} C_DIS
LIN {X -0.348,Y -590.056,Z 1465.170,A 0.000,B 0.000,C 90.000,E1 66.613} C_DIS
LIN {X 0.088,Y -591.064,Z 1465.161,A 0.000,B 0.000,C 90.000,E1 64.973} C_DIS
LIN {X 0.014,Y -592.168,Z 1465.152,A 0.000,B 0.000,C 90.000,E1 63.384} C_DIS
LIN {X 0.127,Y -594.069,Z 1465.137,A 0.000,B 0.000,C 90.000,E1 60.717} C_DIS
LIN {X 0.057,Y -595.683,Z 1465.127,A 0.000,B 0.000,C 90.000,E1 58.869} C_DIS
LIN {X -0.083,Y -597.028,Z 1465.118,A 0.000,B 0.000,C 90.000,E1 57.296} C_DIS
LIN {X 0.176,Y -597.952,Z 1465.112,A 0.000,B 0.000,C 90.000,E1 56.215} C_DIS
LIN {X -0.056,Y -598.863,Z 1465.107,A 0.000,B 0.000,C 90.000,E1 55.182} C_DIS
LIN {X -0.045,Y -599.846,Z 1465.099,A 0.000,B 0.000,C 90.000,E1 53.863} C_DIS
LIN {X -0.130,Y -601.047,Z 1465.089,A 0.000,B 0.000,C 90.000,E1 52.029} C_DIS
LIN {X -0.203,Y -601.961,Z 1465.082,A 0.000,B 0.000,C 90.000,E1 50.723} C_DIS
LIN {X -0.134,Y -602.396,Z 1465.076,A 0.000,B 0.000,C 90.000,E1 49.666} C_DIS
LIN {X 0.224,Y -602.806,Z 1465.066,A 0.000,B 0.000,C 90.000,E1 47.796} C_DIS
LIN {X -0.151,Y -602.977,Z 1465.060,A 0.000,B 0.000,C 90.000,E1 46.782} C_DIS
LIN {X -0.307,Y -602.970,Z 1465.053,A 0.000,B 0.000,C 90.000,E1 45.486} C_DIS
LIN {X 0.392,Y -602.487,Z 1465.045,A 0.000,B 0.000,C 90.000,E1 44.109} C_DIS
LIN {X -0.218,Y -602.054,Z 1465.041,A 0.000,B 0.000,C 90.000,E1 43.380} C_DIS
LIN {X 0.037,Y -601.067,Z 1465.034,A 0.000,B 0.000,C 90.000,E1 42.043} C_DIS
LIN {X 0.299,Y -600.301,Z 1465.029,A 0.000,B 0.000,C 90.000,E1 41.229} C_DIS
LIN {X -0.115,Y -599.115,Z 1465.023,A 0.000,B 0.000,C 90.000,E1 40.216} C_DIS
LIN {X -0.012,Y -597.676,Z 1465.018,A 0.000,B 0.000,C 90.000,E1 39.152} C_DIS
LIN {X 0.221,Y -595.721,Z 1465.010,A 0.000,B 0.000,C 90.000,E1 37.810} C_DIS
LIN {X -0.157,Y -594.905,Z 1465.007,A 0.000,B 0.000,C 90.000,E1 37.317} C_DIS
LIN {X 0.261,Y -592.969,Z 1465.001,A 0.000,B 0.000,C 90.000,E1 36.217} C_DIS
LIN {X 0.081,Y -591.242,Z 1464.997,A 0.000,B 0.000,C 90.000,E1 35.438} C_DIS
LIN {X -0.118,Y -589.362,Z 1464.993,A 0.000,B 0.000,C 90.000,E1 34.659} C_DIS
LIN {X 0.203,Y -585.683,Z 1464.985,A 0.000,B 0.000,C 90.000,E1 33.293} C_DIS
LIN {X 0.116,Y -583.202,Z 1464.981,A 0.000,B 0.000,C 90.000,E1 32.498} C_DIS
LIN {X 0.151,Y -581.321,Z 1464.978,A 0.000,B 0.000,C 90.000,E1 31.957} C_DIS
LIN {X 0.328,Y -578.257,Z 1464.973,A 0.000,B 0.000,C 90.000,E1 31.131} C_DIS
LIN {X 0.171,Y -574.875,Z 1464.969,A 0.000,B 0.000,C 90.000,E1 30.335} C_DIS
LIN {X 0.141,Y -572.346,Z 1464.966,A 0.000,B 0.000,C 90.000,E1 29.795} C_DIS
LIN {X -0.086,Y -568.101,Z 1464.961,A 0.000,B 0.000,C 90.000,E1 28.999} C_DIS
LIN {X 0.138,Y -563.600,Z 1464.957,A 0.000,B 0.000,C 90.000,E1 28.153} C_DIS
LIN {X 0.053,Y -558.639,Z 1464.952,A 0.000,B 0.000,C 90.000,E1 27.334} C_DIS
LIN {X -0.106,Y -555.120,Z 1464.949,A 0.000,B 0.000,C 90.000,E1 26.796} C_DIS
LIN {X -0.273,Y -549.474,Z 1464.944,A 0.000,B 0.000,C 90.000,E1 25.976} C_DIS
LIN {X -0.021,Y -541.134,Z 1464.938,A 0.000,B 0.000,C 90.000,E1 24.823} C_DIS
LIN {X -0.058,Y -536.640,Z 1464.935,A 0.000,B 0.000,C 90.000,E1 24.259} C_DIS
LIN {X -0.077,Y -528.230,Z 1464.929,A 0.000,B 0.000,C 90.000,E1 23.259} C_DIS
LIN {X 0.140,Y -521.847,Z 1464.925,A 0.000,B 0.000,C 90.000,E1 22.514} C_DIS
LIN {X 0.235,Y -517.895,Z 1464.923,A 0.000,B 0.000,C 90.000,E1 22.078} C_DIS
LIN {X -0.259,Y -513.529,Z 1464.921,A 0.000,B 0.000,C 90.000,E1 21.716} C_DIS
LIN {X 0.270,Y -508.655,Z 1464.918,A 0.000,B 0.000,C 90.000,E1 21.280} C_DIS
LIN {X -0.096,Y -505.000,Z 1464.917,A 0.000,B 0.000,C 90.000,E1 21.099} C_DIS
LIN {X -0.103,Y -502.154,Z 1464.917,A 0.000,B 0.000,C 90.000,E1 20.972} C_DIS
LIN {X -0.097,Y -500.034,Z 1464.916,A 0.000,B 0.000,C 90.000,E1 20.918} C_DIS
LIN {X -0.128,Y -499.634,Z 1464.916,A 0.000,B 0.000,C 90.000,E1 20.918} C_DIS
LIN {X -0.120,Y -377.096,Z 1464.916,A 0.000,B 0.000,C 90.000,E1 20.918} C_DIS
LIN {X 0.169,Y -373.668,Z 1464.897,A 0.000,B 0.000,C 90.000,E1 17.511} C_DIS
LIN {X 0.196,Y -368.065,Z 1464.869,A 0.000,B 0.000,C 90.000,E1 12.355} C_DIS
LIN {X 0.006,Y -366.378,Z 1464.854,A 0.000,B 0.000,C 90.000,E1 9.792} C_DIS
LIN {X -0.055,Y -361.730,Z 1464.821,A 0.000,B 0.000,C 90.000,E1 3.841} C_DIS
LIN {X -0.170,Y -360.848,Z 1464.801,A 0.000,B 0.000,C 90.000,E1 0.115} C_DIS
LIN {X -0.053,Y -359.426,Z 1464.770,A 0.000,B 0.000,C 90.000,E1 354.546} C_DIS
LIN {X 0.070,Y -358.890,Z 1464.759,A 0.000,B 0.000,C 90.000,E1 352.648} C_DIS
LIN {X -0.020,Y -359.563,Z 1464.726,A 0.000,B 0.000,C 90.000,E1 346.645} C_DIS
LIN {X 0.001,Y -361.801,Z 1464.684,A 0.000,B 0.000,C 90.000,E1 339.135} C_DIS
LIN {X -0.154,Y -362.053,Z 1464.680,A 0.000,B 0.000,C 90.000,E1 338.411} C_DIS
LIN {X 0.189,Y -365.980,Z 1464.643,A 0.000,B 0.000,C 90.000,E1 331.641} C_DIS
LIN {X 0.029,Y -366.387,Z 1464.639,A 0.000,B 0.000,C 90.000,E1 330.923} C_DIS
LIN {X -0.031,Y -371.355,Z 1464.604,A 0.000,B 0.000,C 90.000,E1 324.642} C_DIS
LIN {X -0.043,Y -371.766,Z 1464.602,A 0.000,B 0.000,C 90.000,E1 324.276} C_DIS
LIN {X 0.013,Y -377.358,Z 1464.567,A 0.000,B 0.000,C 90.000,E1 318.038} C_DIS
LIN {X 0.012,Y -378.235,Z 1464.563,A 0.000,B 0.000,C 90.000,E1 317.310} C_DIS
LIN {X 0.002,Y -383.940,Z 1464.531,A 0.000,B 0.000,C 90.000,E1 311.515} C_DIS
LIN {X 0.088,Y -384.893,Z 1464.527,A 0.000,B 0.000,C 90.000,E1 310.782} C_DIS
LIN {X 0.262,Y -390.610,Z 1464.495,A 0.000,B 0.000,C 90.000,E1 305.025} C_DIS
LIN {X 0.106,Y -391.104,Z 1464.493,A 0.000,B 0.000,C 90.000,E1 304.692} C_DIS
LIN {X 0.022,Y -391.648,Z 1464.489,A 0.000,B 0.000,C 90.000,E1 303.992} C_DIS
LIN {X -0.080,Y -396.825,Z 1464.459,A 0.000,B 0.000,C 90.000,E1 298.693} C_DIS
LIN {X -0.210,Y -397.120,Z 1464.457,A 0.000,B 0.000,C 90.000,E1 298.359} C_DIS
LIN {X -0.055,Y -401.597,Z 1464.426,A 0.000,B 0.000,C 90.000,E1 292.717} C_DIS
LIN {X 0.222,Y -404.659,Z 1464.395,A 0.000,B 0.000,C 90.000,E1 287.094} C_DIS
LIN {X -0.079,Y -404.735,Z 1464.391,A 0.000,B 0.000,C 90.000,E1 286.441} C_DIS
LIN {X 0.214,Y -406.099,Z 1464.364,A 0.000,B 0.000,C 90.000,E1 281.535} C_DIS
LIN {X -0.176,Y -406.094,Z 1464.362,A 0.000,B 0.000,C 90.000,E1 281.243} C_DIS
LIN {X -0.097,Y -405.680,Z 1464.333,A 0.000,B 0.000,C 90.000,E1 276.024} C_DIS
LIN {X -0.165,Y -405.058,Z 1464.328,A 0.000,B 0.000,C 90.000,E1 274.992} C_DIS
LIN {X -0.060,Y -403.497,Z 1464.304,A 0.000,B 0.000,C 90.000,E1 270.802} C_DIS
LIN {X -0.092,Y -403.288,Z 1464.302,A 0.000,B 0.000,C 90.000,E1 270.458} C_DIS
LIN {X 0.091,Y -398.931,Z 1464.271,A 0.000,B 0.000,C 90.000,E1 264.837} C_DIS
LIN {X -0.040,Y -393.108,Z 1464.242,A 0.000,B 0.000,C 90.000,E1 259.567} C_DIS
LIN {X -0.079,Y -392.835,Z 1464.240,A 0.000,B 0.000,C 90.000,E1 259.218} C_DIS
LIN {X 0.034,Y -385.993,Z 1464.212,A 0.000,B 0.000,C 90.000,E1 254.212} C_DIS
LIN {X -0.026,Y -385.267,Z 1464.208,A 0.000,B 0.000,C 90.000,E1 253.504} C_DIS
LIN {X -0.004,Y -384.768,Z 1464.206,A 0.000,B 0.000,C 90.000,E1 253.142} C_DIS
LIN {X 0.221,Y -377.973,Z 1464.182,A 0.000,B 0.000,C 90.000,E1 248.773} C_DIS
LIN {X -0.044,Y -376.233,Z 1464.174,A 0.000,B 0.000,C 90.000,E1 247.358} C_DIS
LIN {X 0.057,Y -374.944,Z 1464.170,A 0.000,B 0.000,C 90.000,E1 246.613} C_DIS
LIN {X -0.208,Y -368.417,Z 1464.148,A 0.000,B 0.000,C 90.000,E1 242.615} C_DIS
LIN {X 0.097,Y -366.047,Z 1464.137,A 0.000,B 0.000,C 90.000,E1 240.717} C_DIS
LIN {X 0.004,Y -359.196,Z 1464.115,A 0.000,B 0.000,C 90.000,E1 236.628} C_DIS
LIN {X 0.021,Y -355.842,Z 1464.100,A 0.000,B 0.000,C 90.000,E1 233.989} C_DIS
LIN {X -0.173,Y -348.793,Z 1464.075,A 0.000,B 0.000,C 90.000,E1 229.461} C_DIS
LIN {X -0.097,Y -346.185,Z 1464.062,A 0.000,B 0.000,C 90.000,E1 227.148} C_DIS
LIN {X -0.088,Y -345.065,Z 1464.058,A 0.000,B 0.000,C 90.000,E1 226.377} C_DIS
LIN {X 0.094,Y -338.586,Z 1464.030,A 0.000,B 0.000,C 90.000,E1 221.310} C_DIS
LIN {X 0.094,Y -336.840,Z 1464.019,A 0.000,B 0.000,C 90.000,E1 219.358} C_DIS
LIN {X 0.014,Y -330.861,Z 1463.988,A 0.000,B 0.000,C 90.000,E1 213.865} C_DIS
LIN {X 0.149,Y -329.296,Z 1463.975,A 0.000,B 0.000,C 90.000,E1 211.465} C_DIS
LIN {X -0.154,Y -324.669,Z 1463.942,A 0.000,B 0.000,C 90.000,E1 205.540} C_DIS
LIN {X 0.174,Y -323.837,Z 1463.928,A 0.000,B 0.000,C 90.000,E1 203.078} C_DIS
LIN {X -0.017,Y -321.124,Z 1463.881,A 0.000,B 0.000,C 90.000,E1 194.662} C_DIS
LIN {X 0.138,Y -320.932,Z 1463.877,A 0.000,B 0.000,C 90.000,E1 193.828} C_DIS
LIN {X -0.076,Y -321.562,Z 1463.832,A 0.000,B 0.000,C 90.000,E1 185.796} C_DIS
LIN {X -0.143,Y -324.415,Z 1463.790,A 0.000,B 0.000,C 90.000,E1 178.165} C_DIS
LIN {X -0.141,Y -325.376,Z 1463.783,A 0.000,B 0.000,C 90.000,E1 176.963} C_DIS
LIN {X -0.100,Y -329.112,Z 1463.750,A 0.000,B 0.000,C 90.000,E1 170.971} C_DIS
LIN {X 0.061,Y -334.260,Z 1463.726,A 0.000,B 0.000,C 90.000,E1 166.589} C_DIS
LIN {X 0.067,Y -335.488,Z 1463.719,A 0.000,B 0.000,C 90.000,E1 165.408} C_DIS
LIN {X 0.143,Y -340.932,Z 1463.695,A 0.000,B 0.000,C 90.000,E1 161.094} C_DIS
LIN {X -0.172,Y -342.138,Z 1463.691,A 0.000,B 0.000,C 90.000,E1 160.369} C_DIS
LIN {X 0.158,Y -345.871,Z 1463.675,A 0.000,B 0.000,C 90.000,E1 157.411} C_DIS
LIN {X 0.171,Y -454.016,Z 1463.675,A 0.000,B 0.000,C 90.000,E1 157.411} C_DIS
LIN {X 0.222,Y -456.619,Z 1463.674,A 0.000,B 0.000,C 90.000,E1 157.358} C_DIS
LIN {X 0.128,Y -460.447,Z 1463.674,A 0.000,B 0.000,C 90.000,E1 157.230} C_DIS
LIN {X 0.028,Y -463.311,Z 1463.673,A 0.000,B 0.000,C 90.000,E1 157.102} C_DIS
LIN {X 0.129,Y -466.279,Z 1463.672,A 0.000,B 0.000,C 90.000,E1 156.922} C_DIS
LIN {X -0.016,Y -472.215,Z 1463.670,A 0.000,B 0.000,C 90.000,E1 156.538} C_DIS
LIN {X 0.084,Y -476.625,Z 1463.668,A 0.000,B 0.000,C 90.000,E1 156.177} C_DIS
LIN {X 0.067,Y -483.930,Z 1463.664,A 0.000,B 0.000,C 90.000,E1 155.537} C_DIS
LIN {X -0.076,Y -491.089,Z 1463.661,A 0.000,B 0.000,C 90.000,E1 154.897} C_DIS
LIN {X 0.118,Y -497.948,Z 1463.657,A 0.000,B 0.000,C 90.000,E1 154.204} C_DIS
LIN {X 0.278,Y -501.992,Z 1463.655,A 0.000,B 0.000,C 90.000,E1 153.768} C_DIS
LIN {X 0.173,Y -507.153,Z 1463.651,A 0.000,B 0.000,C 90.000,E1 153.204} C_DIS
LIN {X -0.104,Y -510.919,Z 1463.649,A 0.000,B 0.000,C 90.000,E1 152.794} C_DIS
LIN {X 0.093,Y -515.417,Z 1463.646,A 0.000,B 0.000,C 90.000,E1 152.180} C_DIS
LIN {X 0.104,Y -519.483,Z 1463.642,A 0.000,B 0.000,C 90.000,E1 151.591} C_DIS
LIN {X 0.147,Y -523.081,Z 1463.639,A 0.000,B 0.000,C 90.000,E1 151.001} C_DIS
LIN {X 0.059,Y -527.069,Z 1463.635,A 0.000,B 0.000,C 90.000,E1 150.284} C_DIS
LIN {X 0.044,Y -531.774,Z 1463.629,A 0.000,B 0.000,C 90.000,E1 149.282} C_DIS
LIN {X 0.016,Y -533.031,Z 1463.628,A 0.000,B 0.000,C 90.000,E1 148.997} C_DIS
LIN {X 0.144,Y -536.322,Z 1463.623,A 0.000,B 0.000,C 90.000,E1 148.122} C_DIS
LIN {X -0.148,Y -537.389,Z 1463.621,A 0.000,B 0.000,C 90.000,E1 147.867} C_DIS
LIN {X 0.020,Y -540.121,Z 1463.617,A 0.000,B 0.000,C 90.000,E1 146.993} C_DIS
LIN {X -0.216,Y -543.444,Z 1463.610,A 0.000,B 0.000,C 90.000,E1 145.881} C_DIS
LIN {X -0.126,Y -545.664,Z 1463.606,A 0.000,B 0.000,C 90.000,E1 145.022} C_DIS
LIN {X -0.323,Y -547.628,Z 1463.601,A 0.000,B 0.000,C 90.000,E1 144.196} C_DIS
LIN {X -0.129,Y -549.904,Z 1463.595,A 0.000,B 0.000,C 90.000,E1 143.050} C_DIS
LIN {X 0.099,Y -551.813,Z 1463.589,A 0.000,B 0.000,C 90.000,E1 141.904} C_DIS
LIN {X -0.148,Y -553.045,Z 1463.584,A 0.000,B 0.000,C 90.000,E1 141.090} C_DIS
LIN {X -0.315,Y -554.431,Z 1463.578,A 0.000,B 0.000,C 90.000,E1 139.989} C_DIS
LIN {X -0.040,Y -555.946,Z 1463.570,A 0.000,B 0.000,C 90.000,E1 138.566} C_DIS
LIN {X -0.124,Y -557.521,Z 1463.561,A 0.000,B 0.000,C 90.000,E1 136.905} C_DIS
LIN {X 0.168,Y -558.683,Z 1463.553,A 0.000,B 0.000,C 90.000,E1 135.486} C_DIS
LIN {X 0.078,Y -559.637,Z 1463.545,A 0.000,B 0.000,C 90.000,E1 134.109} C_DIS
LIN {X -0.006,Y -560.371,Z 1463.537,A 0.000,B 0.000,C 90.000,E1 132.732} C_DIS
LIN {X 0.281,Y -560.721,Z 1463.531,A 0.000,B 0.000,C 90.000,E1 131.595} C_DIS
LIN {X -0.121,Y -560.969,Z 1463.524,A 0.000,B 0.000,C 90.000,E1 130.253} C_DIS
LIN {X -0.068,Y -561.078,Z 1463.514,A 0.000,B 0.000,C 90.000,E1 128.588} C_DIS
LIN {X -0.276,Y -561.222,Z 1463.505,A 0.000,B 0.000,C 90.000,E1 126.950} C_DIS
LIN {X 0.115,Y -561.201,Z 1463.499,A 0.000,B 0.000,C 90.000,E1 125.804} C_DIS
LIN {X 0.082,Y -561.048,Z 1463.494,A 0.000,B 0.000,C 90.000,E1 124.978} C_DIS
LIN {X -0.012,Y -560.468,Z 1463.481,A 0.000,B 0.000,C 90.000,E1 122.498} C_DIS
LIN {X -0.101,Y -560.381,Z 1463.471,A 0.000,B 0.000,C 90.000,E1 120.846} C_DIS
LIN {X -0.007,Y -560.592,Z 1463.461,A 0.000,B 0.000,C 90.000,E1 118.899} C_DIS
LIN {X -0.087,Y -561.046,Z 1463.448,A 0.000,B 0.000,C 90.000,E1 116.693} C_DIS
LIN {X 0.091,Y -561.663,Z 1463.436,A 0.000,B 0.000,C 90.000,E1 114.463} C_DIS
LIN {X -0.079,Y -562.231,Z 1463.427,A 0.000,B 0.000,C 90.000,E1 112.823} C_DIS
LIN {X 0.051,Y -562.780,Z 1463.418,A 0.000,B 0.000,C 90.000,E1 111.153} C_DIS
LIN {X -0.012,Y -563.186,Z 1463.408,A 0.000,B 0.000,C 90.000,E1 109.504} C_DIS
LIN {X -0.033,Y -563.617,Z 1463.401,A 0.000,B 0.000,C 90.000,E1 108.127} C_DIS
LIN {X -0.260,Y -564.058,Z 1463.392,A 0.000,B 0.000,C 90.000,E1 106.496} C_DIS
LIN {X 0.213,Y -564.748,Z 1463.379,A 0.000,B 0.000,C 90.000,E1 104.245} C_DIS
LIN {X 0.024,Y -565.703,Z 1463.367,A 0.000,B 0.000,C 90.000,E1 102.063} C_DIS
LIN {X -0.235,Y -566.286,Z 1463.359,A 0.000,B 0.000,C 90.000,E1 100.715} C_DIS
LIN {X -0.034,Y -566.866,Z 1463.352,A 0.000,B 0.000,C 90.000,E1 99.321} C_DIS
LIN {X -0.124,Y -567.576,Z 1463.341,A 0.000,B 0.000,C 90.000,E1 97.409} C_DIS
LIN {X -0.164,Y -568.821,Z 1463.329,A 0.000,B 0.000,C 90.000,E1 95.220} C_DIS
LIN {X 0.193,Y -570.180,Z 1463.318,A 0.000,B 0.000,C 90.000,E1 93.269} C_DIS
LIN {X 0.147,Y -571.815,Z 1463.306,A 0.000,B 0.000,C 90.000,E1 91.088} C_DIS
LIN {X -0.029,Y -573.378,Z 1463.296,A 0.000,B 0.000,C 90.000,E1 89.198} C_DIS
LIN {X -0.156,Y -574.919,Z 1463.285,A 0.000,B 0.000,C 90.000,E1 87.306} C_DIS
LIN {X 0.209,Y -576.261,Z 1463.276,A 0.000,B 0.000,C 90.000,E1 85.641} C_DIS
LIN {X 0.024,Y -577.650,Z 1463.267,A 0.000,B 0.000,C 90.000,E1 84.033} C_DIS
LIN {X 0.127,Y -579.323,Z 1463.256,A 0.000,B 0.000,C 90.000,E1 82.129} C_DIS
LIN {X -0.224,Y -581.058,Z 1463.246,A 0.000,B 0.000,C 90.000,E1 80.274} C_DIS
LIN {X 0.253,Y -582.799,Z 1463.235,A 0.000,B 0.000,C 90.000,E1 78.342} C_DIS
LIN {X -0.026,Y -584.246,Z 1463.226,A 0.000,B 0.000,C 90.000,E1 76.756} C_DIS
LIN {X -0.201,Y -585.111,Z 1463.220,A 0.000,B 0.000,C 90.000,E1 75.700} C_DIS
LIN {X -0.220,Y -585.771,Z 1463.214,A 0.000,B 0.000,C 90.000,E1 74.629} C_DIS
LIN {X 0.086,Y -586.875,Z 1463.204,A 0.000,B 0.000,C 90.000,E1 72.725} C_DIS
LIN {X -0.065,Y -587.569,Z 1463.197,A 0.000,B 0.000,C 90.000,E1 71.402} C_DIS
LIN {X -0.016,Y -588.349,Z 1463.189,A 0.000,B 0.000,C 90.000,E1 70.061} C_DIS
LIN {X 0.357,Y -589.351,Z 1463.179,A 0.000,B 0.000,C 90.000,E1 68.156} C_DIS
LIN {X -0.230,Y -590.203,Z 1463.170,A 0.000,B 0.000,C 90.000,E1 66.613} C_DIS
LIN {X 0.209,Y -591.228,Z 1463.161,A 0.000,B 0.000,C 90.000,E1 64.973} C_DIS
LIN {X 0.139,Y -592.333,Z 1463.152,A 0.000,B 0.000,C 90.000,E1 63.384} C_DIS
LIN {X 0.259,Y -594.231,Z 1463.137,A 0.000,B 0.000,C 90.000,E1 60.717} C_DIS
LIN {X -0.018,Y -595.637,Z 1463.129,A 0.000,B 0.000,C 90.000,E1 59.154} C_DIS
LIN {X -0.167,Y -597.007,Z 1463.120,A 0.000,B 0.000,C 90.000,E1 57.582} C_DIS
LIN {X 0.319,Y -598.130,Z 1463.113,A 0.000,B 0.000,C 90.000,E1 56.215} C_DIS
LIN {X 0.088,Y -599.052,Z 1463.107,A 0.000,B 0.000,C 90.000,E1 55.182} C_DIS
LIN {X -0.137,Y -600.215,Z 1463.098,A 0.000,B 0.000,C 90.000,E1 53.623} C_DIS
LIN {X -0.099,Y -601.442,Z 1463.088,A 0.000,B 0.000,C 90.000,E1 51.778} C_DIS
LIN {X 0.204,Y -602.313,Z 1463.080,A 0.000,B 0.000,C 90.000,E1 50.436} C_DIS
LIN {X 0.027,Y -602.626,Z 1463.076,A 0.000,B 0.000,C 90.000,E1 49.666} C_DIS
LIN {X 0.148,Y -602.972,Z 1463.067,A 0.000,B 0.000,C 90.000,E1 48.081} C_DIS
LIN {X 0.017,Y -603.230,Z 1463.060,A 0.000,B 0.000,C 90.000,E1 46.782} C_DIS
LIN {X 0.066,Y -603.253,Z 1463.054,A 0.000,B 0.000,C 90.000,E1 45.729} C_DIS
LIN {X 0.118,Y -602.967,Z 1463.048,A 0.000,B 0.000,C 90.000,E1 44.676} C_DIS
LIN {X 0.166,Y -602.502,Z 1463.042,A 0.000,B 0.000,C 90.000,E1 43.623} C_DIS
LIN {X -0.182,Y -601.361,Z 1463.034,A 0.000,B 0.000,C 90.000,E1 42.081} C_DIS
LIN {X 0.057,Y -600.022,Z 1463.026,A 0.000,B 0.000,C 90.000,E1 40.744} C_DIS
LIN {X -0.072,Y -599.091,Z 1463.022,A 0.000,B 0.000,C 90.000,E1 39.967} C_DIS
LIN {X -0.044,Y -596.851,Z 1463.013,A 0.000,B 0.000,C 90.000,E1 38.382} C_DIS
LIN {X 0.044,Y -595.229,Z 1463.007,A 0.000,B 0.000,C 90.000,E1 37.317} C_DIS
LIN {X 0.116,Y -593.304,Z 1463.001,A 0.000,B 0.000,C 90.000,E1 36.251} C_DIS
LIN {X -0.054,Y -591.620,Z 1462.997,A 0.000,B 0.000,C 90.000,E1 35.471} C_DIS
LIN {X -0.242,Y -589.760,Z 1462.993,A 0.000,B 0.000,C 90.000,E1 34.692} C_DIS
LIN {X -0.392,Y -586.131,Z 1462.985,A 0.000,B 0.000,C 90.000,E1 33.372} C_DIS
LIN {X 0.018,Y -582.787,Z 1462.979,A 0.000,B 0.000,C 90.000,E1 32.260} C_DIS
LIN {X -0.097,Y -579.800,Z 1462.975,A 0.000,B 0.000,C 90.000,E1 31.465} C_DIS
LIN {X -0.237,Y -576.575,Z 1462.970,A 0.000,B 0.000,C 90.000,E1 30.669} C_DIS
LIN {X -0.328,Y -573.597,Z 1462.967,A 0.000,B 0.000,C 90.000,E1 30.001} C_DIS
LIN {X -0.038,Y -569.447,Z 1462.962,A 0.000,B 0.000,C 90.000,E1 29.155} C_DIS
LIN {X 0.116,Y -564.267,Z 1462.957,A 0.000,B 0.000,C 90.000,E1 28.180} C_DIS
LIN {X -0.295,Y -558.494,Z 1462.951,A 0.000,B 0.000,C 90.000,E1 27.257} C_DIS
LIN {X -0.067,Y -554.040,Z 1462.948,A 0.000,B 0.000,C 90.000,E1 26.539} C_DIS
LIN {X -0.129,Y -549.290,Z 1462.944,A 0.000,B 0.000,C 90.000,E1 25.848} C_DIS
LIN {X 0.018,Y -542.020,Z 1462.938,A 0.000,B 0.000,C 90.000,E1 24.847} C_DIS
LIN {X 0.213,Y -537.602,Z 1462.935,A 0.000,B 0.000,C 90.000,E1 24.259} C_DIS
LIN {X 0.006,Y -531.603,Z 1462.931,A 0.000,B 0.000,C 90.000,E1 23.567} C_DIS
LIN {X 0.078,Y -524.188,Z 1462.926,A 0.000,B 0.000,C 90.000,E1 22.695} C_DIS
LIN {X 0.066,Y -515.307,Z 1462.921,A 0.000,B 0.000,C 90.000,E1 21.716} C_DIS
LIN {X 0.187,Y -510.919,Z 1462.918,A 0.000,B 0.000,C 90.000,E1 21.280} C_DIS
LIN {X -0.071,Y -507.848,Z 1462.917,A 0.000,B 0.000,C 90.000,E1 21.046} C_DIS
LIN {X 0.068,Y -502.936,Z 1462.915,A 0.000,B 0.000,C 90.000,E1 20.663} C_DIS
LIN {X 0.042,Y -501.123,Z 1462.914,A 0.000,B 0.000,C 90.000,E1 20.556} C_DIS
LIN {X -0.234,Y -497.862,Z 1462.913,A 0.000,B 0.000,C 90.000,E1 20.429} C_DIS
LIN {X -0.153,Y -495.718,Z 1462.913,A 0.000,B 0.000,C 90.000,E1 20.355} C_DIS
LIN {X 0.218,Y -494.960,Z 1462.913,A 0.000,B 0.000,C 90.000,E1 20.301} C_DIS
LIN {X 0.142,Y -376.409,Z 1462.913,A 0.000,B 0.000,C 90.000,E1 20.301} C_DIS
LIN {X 0.040,Y -373.458,Z 1462.896,A 0.000,B 0.000,C 90.000,E1 17.347} C_DIS
LIN {X 0.084,Y -367.921,Z 1462.868,A 0.000,B 0.000,C 90.000,E1 12.187} C_DIS
LIN {X 0.105,Y -366.514,Z 1462.855,A 0.000,B 0.000,C 90.000,E1 9.962} C_DIS
LIN {X 0.039,Y -361.812,Z 1462.822,A 0.000,B 0.000,C 90.000,E1 4.012} C_DIS
LIN {X -0.076,Y -360.904,Z 1462.802,A 0.000,B 0.000,C 90.000,E1 0.286} C_DIS
LIN {X -0.053,Y -359.426,Z 1462.770,A 0.000,B 0.000,C 90.000,E1 354.546} C_DIS
LIN {X 0.070,Y -358.890,Z 1462.759,A 0.000,B 0.000,C 90.000,E1 352.648} C_DIS
LIN {X -0.020,Y -359.563,Z 1462.726,A 0.000,B 0.000,C 90.000,E1 346.645} C_DIS
LIN {X 0.001,Y -361.801,Z 1462.684,A 0.000,B 0.000,C 90.000,E1 339.135} C_DIS
LIN {X -0.154,Y -362.053,Z 1462.680,A 0.000,B 0.000,C 90.000,E1 338.411} C_DIS
LIN {X 0.189,Y -365.980,Z 1462.643,A 0.000,B 0.000,C 90.000,E1 331.641} C_DIS
LIN {X 0.029,Y -366.387,Z 1462.639,A 0.000,B 0.000,C 90.000,E1 330.923} C_DIS
LIN {X -0.031,Y -371.355,Z 1462.604,A 0.000,B 0.000,C 90.000,E1 324.642} C_DIS
LIN {X -0.043,Y -371.766,Z 1462.602,A 0.000,B 0.000,C 90.000,E1 324.276} C_DIS
LIN {X 0.013,Y -377.358,Z 1462.567,A 0.000,B 0.000,C 90.000,E1 318.038} C_DIS
LIN {X 0.012,Y -378.235,Z 1462.563,A 0.000,B 0.000,C 90.000,E1 317.310} C_DIS
LIN {X 0.002,Y -383.940,Z 1462.531,A 0.000,B 0.000,C 90.000,E1 311.515} C_DIS
LIN {X 0.088,Y -384.893,Z 1462.527,A 0.000,B 0.000,C 90.000,E1 310.782} C_DIS
LIN {X 0.262,Y -390.610,Z 1462.495,A 0.000,B 0.000,C 90.000,E1 305.025} C_DIS
LIN {X 0.106,Y -391.104,Z 1462.493,A 0.000,B 0.000,C 90.000,E1 304.692} C_DIS
LIN {X 0.022,Y -391.648,Z 1462.489,A 0.000,B 0.000,C 90.000,E1 303.992} C_DIS
LIN {X -0.080,Y -396.825,Z 1462.459,A 0.000,B 0.000,C 90.000,E1 298.693} C_DIS
LIN {X -0.210,Y -397.120,Z 1462.457,A 0.000,B 0.000,C 90.000,E1 298.359} C_DIS
LIN {X -0.055,Y -401.597,Z 1462.426,A 0.000,B 0.000,C 90.000,E1 292.717} C_DIS
LIN {X 0.222,Y -404.659,Z 1462.395,A 0.000,B 0.000,C 90.000,E1 287.094} C_DIS
LIN {X -0.079,Y -404.735,Z 1462.391,A 0.000,B 0.000,C 90.000,E1 286.441} C_DIS
LIN {X 0.214,Y -406.099,Z 1462.364,A 0.000,B 0.000,C 90.000,E1 281.535} C_DIS
LIN {X -0.176,Y -406.094,Z 1462.362,A 0.000,B 0.000,C 90.000,E1 281.243} C_DIS
LIN {X -0.097,Y -405.680,Z 1462.333,A 0.000,B 0.000,C 90.000,E1 276.024} C_DIS
LIN {X -0.165,Y -405.058,Z 1462.328,A 0.000,B 0.000,C 90.000,E1 274.992} C_DIS
LIN {X -0.060,Y -403.497,Z 1462.304,A 0.000,B 0.000,C 90.000,E1 270.802} C_DIS
LIN {X -0.092,Y -403.288,Z 1462.302,A 0.000,B 0.000,C 90.000,E1 270.458} C_DIS
LIN {X 0.091,Y -398.931,Z 1462.271,A 0.000,B 0.000,C 90.000,E1 264.837} C_DIS
LIN {X -0.040,Y -393.108,Z 1462.242,A 0.000,B 0.000,C 90.000,E1 259.567} C_DIS
LIN {X -0.079,Y -392.835,Z 1462.240,A 0.000,B 0.000,C 90.000,E1 259.218} C_DIS
LIN {X 0.034,Y -385.993,Z 1462.212,A 0.000,B 0.000,C 90.000,E1 254.212} C_DIS
LIN {X -0.026,Y -385.267,Z 1462.208,A 0.000,B 0.000,C 90.000,E1 253.504} C_DIS
LIN {X -0.004,Y -384.768,Z 1462.206,A 0.000,B 0.000,C 90.000,E1 253.142} C_DIS
LIN {X 0.221,Y -377.973,Z 1462.182,A 0.000,B 0.000,C 90.000,E1 248.773} C_DIS
LIN {X -0.044,Y -376.233,Z 1462.174,A 0.000,B 0.000,C 90.000,E1 247.358} C_DIS
LIN {X 0.057,Y -374.944,Z 1462.170,A 0.000,B 0.000,C 90.000,E1 246.613} C_DIS
LIN {X -0.208,Y -368.417,Z 1462.148,A 0.000,B 0.000,C 90.000,E1 242.615} C_DIS
LIN {X 0.097,Y -366.047,Z 1462.137,A 0.000,B 0.000,C 90.000,E1 240.717} C_DIS
LIN {X 0.004,Y -359.196,Z 1462.115,A 0.000,B 0.000,C 90.000,E1 236.628} C_DIS
LIN {X 0.021,Y -355.842,Z 1462.100,A 0.000,B 0.000,C 90.000,E1 233.989} C_DIS
LIN {X -0.173,Y -348.793,Z 1462.075,A 0.000,B 0.000,C 90.000,E1 229.461} C_DIS
LIN {X -0.097,Y -346.185,Z 1462.062,A 0.000,B 0.000,C 90.000,E1 227.148} C_DIS
LIN {X -0.088,Y -345.065,Z 1462.058,A 0.000,B 0.000,C 90.000,E1 226.377} C_DIS
LIN {X 0.094,Y -338.586,Z 1462.030,A 0.000,B 0.000,C 90.000,E1 221.310} C_DIS
LIN {X 0.094,Y -336.840,Z 1462.019,A 0.000,B 0.000,C 90.000,E1 219.358} C_DIS
LIN {X 0.014,Y -330.861,Z 1461.988,A 0.000,B 0.000,C 90.000,E1 213.865} C_DIS
LIN {X 0.149,Y -329.296,Z 1461.975,A 0.000,B 0.000,C 90.000,E1 211.465} C_DIS
LIN {X -0.154,Y -324.669,Z 1461.942,A 0.000,B 0.000,C 90.000,E1 205.540} C_DIS
LIN {X 0.174,Y -323.837,Z 1461.928,A 0.000,B 0.000,C 90.000,E1 203.078} C_DIS
LIN {X -0.017,Y -321.124,Z 1461.881,A 0.000,B 0.000,C 90.000,E1 194.662} C_DIS
LIN {X 0.138,Y -320.932,Z 1461.877,A 0.000,B 0.000,C 90.000,E1 193.828} C_DIS
LIN {X -0.076,Y -321.562,Z 1461.832,A 0.000,B 0.000,C 90.000,E1 185.796} C_DIS
LIN {X -0.143,Y -324.415,Z 1461.790,A 0.000,B 0.000,C 90.000,E1 178.165} C_DIS
LIN {X -0.141,Y -325.376,Z 1461.783,A 0.000,B 0.000,C 90.000,E1 176.963} C_DIS
LIN {X -0.100,Y -329.112,Z 1461.750,A 0.000,B 0.000,C 90.000,E1 170.971} C_DIS
LIN {X 0.061,Y -334.260,Z 1461.726,A 0.000,B 0.000,C 90.000,E1 166.589} C_DIS
LIN {X 0.067,Y -335.488,Z 1461.719,A 0.000,B 0.000,C 90.000,E1 165.408} C_DIS
LIN {X 0.143,Y -340.932,Z 1461.695,A 0.000,B 0.000,C 90.000,E1 161.094} C_DIS
LIN {X -0.172,Y -342.138,Z 1461.691,A 0.000,B 0.000,C 90.000,E1 160.369} C_DIS
LIN {X 0.183,Y -345.064,Z 1461.678,A 0.000,B 0.000,C 90.000,E1 157.975} C_DIS
LIN {X 0.206,Y -447.936,Z 1461.678,A 0.000,B 0.000,C 90.000,E1 157.975} C_DIS
LIN {X 0.108,Y -448.979,Z 1461.678,A 0.000,B 0.000,C 90.000,E1 157.975} C_DIS
LIN {X -0.014,Y -451.635,Z 1461.677,A 0.000,B 0.000,C 90.000,E1 157.922} C_DIS
LIN {X 0.033,Y -453.474,Z 1461.677,A 0.000,B 0.000,C 90.000,E1 157.847} C_DIS
LIN {X 0.146,Y -457.948,Z 1461.676,A 0.000,B 0.000,C 90.000,E1 157.614} C_DIS
LIN {X -0.265,Y -461.009,Z 1461.675,A 0.000,B 0.000,C 90.000,E1 157.486} C_DIS
LIN {X -0.041,Y -467.020,Z 1461.672,A 0.000,B 0.000,C 90.000,E1 157.050} C_DIS
LIN {X 0.096,Y -472.954,Z 1461.670,A 0.000,B 0.000,C 90.000,E1 156.561} C_DIS
LIN {X 0.137,Y -481.723,Z 1461.666,A 0.000,B 0.000,C 90.000,E1 155.793} C_DIS
LIN {X 0.021,Y -488.945,Z 1461.662,A 0.000,B 0.000,C 90.000,E1 155.153} C_DIS
LIN {X 0.196,Y -495.990,Z 1461.658,A 0.000,B 0.000,C 90.000,E1 154.460} C_DIS
LIN {X -0.137,Y -502.580,Z 1461.655,A 0.000,B 0.000,C 90.000,E1 153.819} C_DIS
LIN {X -0.226,Y -507.706,Z 1461.651,A 0.000,B 0.000,C 90.000,E1 153.256} C_DIS
LIN {X -0.054,Y -511.460,Z 1461.649,A 0.000,B 0.000,C 90.000,E1 152.794} C_DIS
LIN {X -0.309,Y -515.909,Z 1461.646,A 0.000,B 0.000,C 90.000,E1 152.231} C_DIS
LIN {X -0.295,Y -519.960,Z 1461.642,A 0.000,B 0.000,C 90.000,E1 151.641} C_DIS
LIN {X 0.048,Y -524.347,Z 1461.638,A 0.000,B 0.000,C 90.000,E1 150.873} C_DIS
LIN {X -0.175,Y -526.804,Z 1461.636,A 0.000,B 0.000,C 90.000,E1 150.461} C_DIS
LIN {X -0.115,Y -530.945,Z 1461.631,A 0.000,B 0.000,C 90.000,E1 149.587} C_DIS
LIN {X 0.163,Y -532.926,Z 1461.629,A 0.000,B 0.000,C 90.000,E1 149.125} C_DIS
LIN {X 0.148,Y -536.750,Z 1461.623,A 0.000,B 0.000,C 90.000,E1 148.122} C_DIS
LIN {X -0.143,Y -537.807,Z 1461.621,A 0.000,B 0.000,C 90.000,E1 147.867} C_DIS
LIN {X 0.030,Y -540.496,Z 1461.617,A 0.000,B 0.000,C 90.000,E1 146.993} C_DIS
LIN {X -0.200,Y -543.808,Z 1461.610,A 0.000,B 0.000,C 90.000,E1 145.881} C_DIS
LIN {X -0.106,Y -546.019,Z 1461.606,A 0.000,B 0.000,C 90.000,E1 145.022} C_DIS
LIN {X -0.299,Y -547.945,Z 1461.601,A 0.000,B 0.000,C 90.000,E1 144.196} C_DIS
LIN {X -0.100,Y -550.211,Z 1461.595,A 0.000,B 0.000,C 90.000,E1 143.050} C_DIS
LIN {X 0.131,Y -552.085,Z 1461.589,A 0.000,B 0.000,C 90.000,E1 141.904} C_DIS
LIN {X -0.113,Y -553.310,Z 1461.584,A 0.000,B 0.000,C 90.000,E1 141.090} C_DIS
LIN {X -0.276,Y -554.662,Z 1461.578,A 0.000,B 0.000,C 90.000,E1 139.989} C_DIS
LIN {X 0.004,Y -556.145,Z 1461.570,A 0.000,B 0.000,C 90.000,E1 138.566} C_DIS
LIN {X 0.265,Y -557.426,Z 1461.562,A 0.000,B 0.000,C 90.000,E1 137.148} C_DIS
LIN {X -0.235,Y -558.595,Z 1461.554,A 0.000,B 0.000,C 90.000,E1 135.810} C_DIS
LIN {X -0.327,Y -559.583,Z 1461.547,A 0.000,B 0.000,C 90.000,E1 134.433} C_DIS
LIN {X 0.258,Y -560.075,Z 1461.542,A 0.000,B 0.000,C 90.000,E1 133.542} C_DIS
LIN {X 0.129,Y -560.564,Z 1461.536,A 0.000,B 0.000,C 90.000,E1 132.447} C_DIS
LIN {X -0.034,Y -560.811,Z 1461.531,A 0.000,B 0.000,C 90.000,E1 131.634} C_DIS
LIN {X -0.063,Y -561.015,Z 1461.524,A 0.000,B 0.000,C 90.000,E1 130.253} C_DIS
LIN {X 0.086,Y -561.149,Z 1461.513,A 0.000,B 0.000,C 90.000,E1 128.302} C_DIS
LIN {X -0.216,Y -561.247,Z 1461.505,A 0.000,B 0.000,C 90.000,E1 126.950} C_DIS
LIN {X 0.176,Y -561.202,Z 1461.499,A 0.000,B 0.000,C 90.000,E1 125.804} C_DIS
LIN {X 0.143,Y -561.050,Z 1461.495,A 0.000,B 0.000,C 90.000,E1 124.978} C_DIS
LIN {X 0.174,Y -560.543,Z 1461.484,A 0.000,B 0.000,C 90.000,E1 123.038} C_DIS
LIN {X -0.040,Y -560.381,Z 1461.471,A 0.000,B 0.000,C 90.000,E1 120.846} C_DIS
LIN {X 0.122,Y -560.635,Z 1461.459,A 0.000,B 0.000,C 90.000,E1 118.615} C_DIS
LIN {X 0.026,Y -561.117,Z 1461.447,A 0.000,B 0.000,C 90.000,E1 116.411} C_DIS
LIN {X 0.152,Y -561.690,Z 1461.436,A 0.000,B 0.000,C 90.000,E1 114.463} C_DIS
LIN {X -0.018,Y -562.258,Z 1461.427,A 0.000,B 0.000,C 90.000,E1 112.823} C_DIS
LIN {X 0.114,Y -562.796,Z 1461.418,A 0.000,B 0.000,C 90.000,E1 111.153} C_DIS
LIN {X 0.262,Y -563.138,Z 1461.410,A 0.000,B 0.000,C 90.000,E1 109.758} C_DIS
LIN {X -0.111,Y -563.597,Z 1461.402,A 0.000,B 0.000,C 90.000,E1 108.417} C_DIS
LIN {X -0.197,Y -564.111,Z 1461.392,A 0.000,B 0.000,C 90.000,E1 106.496} C_DIS
LIN {X -0.269,Y -564.813,Z 1461.379,A 0.000,B 0.000,C 90.000,E1 104.300} C_DIS
LIN {X 0.093,Y -565.838,Z 1461.367,A 0.000,B 0.000,C 90.000,E1 102.063} C_DIS
LIN {X 0.220,Y -566.344,Z 1461.361,A 0.000,B 0.000,C 90.000,E1 100.950} C_DIS
LIN {X 0.040,Y -566.974,Z 1461.352,A 0.000,B 0.000,C 90.000,E1 99.321} C_DIS
LIN {X 0.173,Y -567.393,Z 1461.344,A 0.000,B 0.000,C 90.000,E1 97.936} C_DIS
LIN {X 0.026,Y -569.016,Z 1461.328,A 0.000,B 0.000,C 90.000,E1 94.935} C_DIS
LIN {X 0.269,Y -570.207,Z 1461.318,A 0.000,B 0.000,C 90.000,E1 93.269} C_DIS
LIN {X 0.224,Y -571.874,Z 1461.306,A 0.000,B 0.000,C 90.000,E1 91.088} C_DIS
LIN {X 0.051,Y -573.437,Z 1461.296,A 0.000,B 0.000,C 90.000,E1 89.198} C_DIS
LIN {X -0.075,Y -574.978,Z 1461.285,A 0.000,B 0.000,C 90.000,E1 87.306} C_DIS
LIN {X 0.147,Y -576.144,Z 1461.277,A 0.000,B 0.000,C 90.000,E1 85.927} C_DIS
LIN {X 0.110,Y -577.744,Z 1461.267,A 0.000,B 0.000,C 90.000,E1 84.033} C_DIS
LIN {X -0.137,Y -578.930,Z 1461.259,A 0.000,B 0.000,C 90.000,E1 82.704} C_DIS
LIN {X -0.140,Y -580.417,Z 1461.250,A 0.000,B 0.000,C 90.000,E1 81.084} C_DIS
LIN {X -0.018,Y -581.921,Z 1461.241,A 0.000,B 0.000,C 90.000,E1 79.454} C_DIS
LIN {X 0.129,Y -583.408,Z 1461.233,A 0.000,B 0.000,C 90.000,E1 77.825} C_DIS
LIN {X 0.313,Y -584.610,Z 1461.225,A 0.000,B 0.000,C 90.000,E1 76.464} C_DIS
LIN {X 0.140,Y -585.425,Z 1461.219,A 0.000,B 0.000,C 90.000,E1 75.408} C_DIS
LIN {X -0.204,Y -586.200,Z 1461.212,A 0.000,B 0.000,C 90.000,E1 74.102} C_DIS
LIN {X 0.192,Y -587.043,Z 1461.204,A 0.000,B 0.000,C 90.000,E1 72.725} C_DIS
LIN {X -0.188,Y -587.605,Z 1461.198,A 0.000,B 0.000,C 90.000,E1 71.692} C_DIS
LIN {X 0.096,Y -588.496,Z 1461.189,A 0.000,B 0.000,C 90.000,E1 70.061} C_DIS
LIN {X 0.136,Y -589.673,Z 1461.177,A 0.000,B 0.000,C 90.000,E1 67.922} C_DIS
LIN {X -0.220,Y -590.509,Z 1461.169,A 0.000,B 0.000,C 90.000,E1 66.357} C_DIS
LIN {X 0.229,Y -591.527,Z 1461.160,A 0.000,B 0.000,C 90.000,E1 64.717} C_DIS
LIN {X 0.265,Y -592.502,Z 1461.152,A 0.000,B 0.000,C 90.000,E1 63.384} C_DIS
LIN {X 0.100,Y -594.392,Z 1461.138,A 0.000,B 0.000,C 90.000,E1 60.745} C_DIS
LIN {X 0.214,Y -595.591,Z 1461.130,A 0.000,B 0.000,C 90.000,E1 59.410} C_DIS
LIN {X -0.028,Y -597.214,Z 1461.120,A 0.000,B 0.000,C 90.000,E1 57.582} C_DIS
LIN {X -0.367,Y -598.310,Z 1461.113,A 0.000,B 0.000,C 90.000,E1 56.294} C_DIS
LIN {X 0.235,Y -599.244,Z 1461.107,A 0.000,B 0.000,C 90.000,E1 55.182} C_DIS
LIN {X 0.014,Y -600.400,Z 1461.098,A 0.000,B 0.000,C 90.000,E1 53.623} C_DIS
LIN {X -0.190,Y -601.478,Z 1461.089,A 0.000,B 0.000,C 90.000,E1 52.065} C_DIS
LIN {X -0.102,Y -602.528,Z 1461.080,A 0.000,B 0.000,C 90.000,E1 50.481} C_DIS
LIN {X -0.412,Y -602.907,Z 1461.075,A 0.000,B 0.000,C 90.000,E1 49.461} C_DIS
LIN {X 0.069,Y -603.117,Z 1461.069,A 0.000,B 0.000,C 90.000,E1 48.366} C_DIS
LIN {X 0.189,Y -603.454,Z 1461.060,A 0.000,B 0.000,C 90.000,E1 46.782} C_DIS
LIN {X 0.240,Y -603.507,Z 1461.054,A 0.000,B 0.000,C 90.000,E1 45.729} C_DIS
LIN {X 0.296,Y -603.234,Z 1461.048,A 0.000,B 0.000,C 90.000,E1 44.676} C_DIS
LIN {X 0.346,Y -602.771,Z 1461.043,A 0.000,B 0.000,C 90.000,E1 43.623} C_DIS
LIN {X 0.005,Y -601.638,Z 1461.034,A 0.000,B 0.000,C 90.000,E1 42.081} C_DIS
LIN {X -0.145,Y -600.317,Z 1461.026,A 0.000,B 0.000,C 90.000,E1 40.782} C_DIS
LIN {X -0.339,Y -599.391,Z 1461.022,A 0.000,B 0.000,C 90.000,E1 40.011} C_DIS
LIN {X 0.154,Y -597.158,Z 1461.013,A 0.000,B 0.000,C 90.000,E1 38.382} C_DIS
LIN {X 0.015,Y -595.965,Z 1461.009,A 0.000,B 0.000,C 90.000,E1 37.604} C_DIS
LIN {X 0.097,Y -594.153,Z 1461.003,A 0.000,B 0.000,C 90.000,E1 36.537} C_DIS
LIN {X 0.282,Y -592.558,Z 1460.999,A 0.000,B 0.000,C 90.000,E1 35.724} C_DIS
LIN {X -0.031,Y -590.154,Z 1460.993,A 0.000,B 0.000,C 90.000,E1 34.692} C_DIS
LIN {X -0.175,Y -586.560,Z 1460.985,A 0.000,B 0.000,C 90.000,E1 33.372} C_DIS
LIN {X -0.071,Y -583.235,Z 1460.979,A 0.000,B 0.000,C 90.000,E1 32.291} C_DIS
LIN {X 0.129,Y -580.309,Z 1460.975,A 0.000,B 0.000,C 90.000,E1 31.465} C_DIS
LIN {X 0.141,Y -578.237,Z 1460.972,A 0.000,B 0.000,C 90.000,E1 30.924} C_DIS
LIN {X 0.135,Y -575.995,Z 1460.969,A 0.000,B 0.000,C 90.000,E1 30.384} C_DIS
LIN {X -0.252,Y -572.873,Z 1460.965,A 0.000,B 0.000,C 90.000,E1 29.745} C_DIS
LIN {X 0.221,Y -567.874,Z 1460.960,A 0.000,B 0.000,C 90.000,E1 28.743} C_DIS
LIN {X -0.229,Y -564.144,Z 1460.956,A 0.000,B 0.000,C 90.000,E1 28.103} C_DIS
LIN {X -0.246,Y -557.500,Z 1460.950,A 0.000,B 0.000,C 90.000,E1 27.001} C_DIS
LIN {X 0.245,Y -551.078,Z 1460.944,A 0.000,B 0.000,C 90.000,E1 25.976} C_DIS
LIN {X 0.158,Y -546.000,Z 1460.941,A 0.000,B 0.000,C 90.000,E1 25.283} C_DIS
LIN {X 0.075,Y -540.713,Z 1460.937,A 0.000,B 0.000,C 90.000,E1 24.591} C_DIS
LIN {X 0.172,Y -537.380,Z 1460.934,A 0.000,B 0.000,C 90.000,E1 24.155} C_DIS
LIN {X -0.028,Y -531.362,Z 1460.930,A 0.000,B 0.000,C 90.000,E1 23.462} C_DIS
LIN {X 0.047,Y -523.915,Z 1460.926,A 0.000,B 0.000,C 90.000,E1 22.589} C_DIS
LIN {X 0.114,Y -513.689,Z 1460.919,A 0.000,B 0.000,C 90.000,E1 21.461} C_DIS
LIN {X 0.047,Y -509.576,Z 1460.917,A 0.000,B 0.000,C 90.000,E1 21.046} C_DIS
LIN {X -0.181,Y -505.206,Z 1460.915,A 0.000,B 0.000,C 90.000,E1 20.663} C_DIS
LIN {X 0.110,Y -500.437,Z 1460.913,A 0.000,B 0.000,C 90.000,E1 20.248} C_DIS
LIN {X 0.310,Y -496.919,Z 1460.911,A 0.000,B 0.000,C 90.000,E1 19.993} C_DIS
LIN {X 0.146,Y -492.957,Z 1460.910,A 0.000,B 0.000,C 90.000,E1 19.812} C_DIS
LIN {X -0.013,Y -490.691,Z 1460.910,A 0.000,B 0.000,C 90.000,E1 19.758} C_DIS
LIN {X -0.141,Y -489.762,Z 1460.910,A 0.000,B 0.000,C 90.000,E1 19.758} C_DIS
LIN {X -0.140,Y -375.753,Z 1460.910,A 0.000,B 0.000,C 90.000,E1 19.758} C_DIS
LIN {X 0.118,Y -373.450,Z 1460.896,A 0.000,B 0.000,C 90.000,E1 17.330} C_DIS
LIN {X 0.051,Y -367.918,Z 1460.868,A 0.000,B 0.000,C 90.000,E1 12.187} C_DIS
LIN {X 0.071,Y -366.512,Z 1460.855,A 0.000,B 0.000,C 90.000,E1 9.962} C_DIS
LIN {X 0.006,Y -361.810,Z 1460.822,A 0.000,B 0.000,C 90.000,E1 4.012} C_DIS
LIN {X -0.108,Y -360.904,Z 1460.802,A 0.000,B 0.000,C 90.000,E1 0.286} C_DIS
LIN {X -0.053,Y -359.426,Z 1460.770,A 0.000,B 0.000,C 90.000,E1 354.546} C_DIS
LIN {X 0.070,Y -358.890,Z 1460.759,A 0.000,B 0.000,C 90.000,E1 352.648} C_DIS
LIN {X -0.020,Y -359.563,Z 1460.726,A 0.000,B 0.000,C 90.000,E1 346.645} C_DIS
LIN {X 0.001,Y -361.801,Z 1460.684,A 0.000,B 0.000,C 90.000,E1 339.135} C_DIS
LIN {X -0.154,Y -362.053,Z 1460.680,A 0.000,B 0.000,C 90.000,E1 338.411} C_DIS
LIN {X 0.189,Y -365.980,Z 1460.643,A 0.000,B 0.000,C 90.000,E1 331.641} C_DIS
LIN {X 0.029,Y -366.387,Z 1460.639,A 0.000,B 0.000,C 90.000,E1 330.923} C_DIS
LIN {X -0.031,Y -371.355,Z 1460.604,A 0.000,B 0.000,C 90.000,E1 324.642} C_DIS
LIN {X -0.043,Y -371.766,Z 1460.602,A 0.000,B 0.000,C 90.000,E1 324.276} C_DIS
LIN {X 0.013,Y -377.358,Z 1460.567,A 0.000,B 0.000,C 90.000,E1 318.038} C_DIS
LIN {X 0.012,Y -378.235,Z 1460.563,A 0.000,B 0.000,C 90.000,E1 317.310} C_DIS
LIN {X 0.002,Y -383.940,Z 1460.531,A 0.000,B 0.000,C 90.000,E1 311.515} C_DIS
LIN {X 0.088,Y -384.893,Z 1460.527,A 0.000,B 0.000,C 90.000,E1 310.782} C_DIS
LIN {X 0.262,Y -390.610,Z 1460.495,A 0.000,B 0.000,C 90.000,E1 305.025} C_DIS
LIN {X 0.106,Y -391.104,Z 1460.493,A 0.000,B 0.000,C 90.000,E1 304.692} C_DIS
LIN {X 0.022,Y -391.648,Z 1460.489,A 0.000,B 0.000,C 90.000,E1 303.992} C_DIS
LIN {X -0.080,Y -396.825,Z 1460.459,A 0.000,B 0.000,C 90.000,E1 298.693} C_DIS
LIN {X -0.210,Y -397.120,Z 1460.457,A 0.000,B 0.000,C 90.000,E1 298.359} C_DIS
LIN {X -0.055,Y -401.597,Z 1460.426,A 0.000,B 0.000,C 90.000,E1 292.717} C_DIS
LIN {X 0.222,Y -404.659,Z 1460.395,A 0.000,B 0.000,C 90.000,E1 287.094} C_DIS
LIN {X -0.079,Y -404.735,Z 1460.391,A 0.000,B 0.000,C 90.000,E1 286.441} C_DIS
LIN {X 0.214,Y -406.099,Z 1460.364,A 0.000,B 0.000,C 90.000,E1 281.535} C_DIS
LIN {X -0.176,Y -406.094,Z 1460.362,A 0.000,B 0.000,C 90.000,E1 281.243} C_DIS
LIN {X -0.097,Y -405.680,Z 1460.333,A 0.000,B 0.000,C 90.000,E1 276.024} C_DIS
LIN {X -0.165,Y -405.058,Z 1460.328,A 0.000,B 0.000,C 90.000,E1 274.992} C_DIS
LIN {X -0.060,Y -403.497,Z 1460.304,A 0.000,B 0.000,C 90.000,E1 270.802} C_DIS
LIN {X -0.092,Y -403.288,Z 1460.302,A 0.000,B 0.000,C 90.000,E1 270.458} C_DIS
LIN {X 0.091,Y -398.931,Z 1460.271,A 0.000,B 0.000,C 90.000,E1 264.837} C_DIS
LIN {X -0.040,Y -393.108,Z 1460.242,A 0.000,B 0.000,C 90.000,E1 259.567} C_DIS
LIN {X -0.079,Y -392.835,Z 1460.240,A 0.000,B 0.000,C 90.000,E1 259.218} C_DIS
LIN {X 0.034,Y -385.993,Z 1460.212,A 0.000,B 0.000,C 90.000,E1 254.212} C_DIS
LIN {X -0.026,Y -385.267,Z 1460.208,A 0.000,B 0.000,C 90.000,E1 253.504} C_DIS
LIN {X -0.004,Y -384.768,Z 1460.206,A 0.000,B 0.000,C 90.000,E1 253.142} C_DIS
LIN {X 0.221,Y -377.973,Z 1460.182,A 0.000,B 0.000,C 90.000,E1 248.773} C_DIS
LIN {X -0.044,Y -376.233,Z 1460.174,A 0.000,B 0.000,C 90.000,E1 247.358} C_DIS
LIN {X 0.057,Y -374.944,Z 1460.170,A 0.000,B 0.000,C 90.000,E1 246.613} C_DIS
LIN {X -0.208,Y -368.417,Z 1460.148,A 0.000,B 0.000,C 90.000,E1 242.615} C_DIS
LIN {X 0.097,Y -366.047,Z 1460.137,A 0.000,B 0.000,C 90.000,E1 240.717} C_DIS
LIN {X 0.004,Y -359.196,Z 1460.115,A 0.000,B 0.000,C 90.000,E1 236.628} C_DIS
LIN {X 0.021,Y -355.842,Z 1460.100,A 0.000,B 0.000,C 90.000,E1 233.989} C_DIS
LIN {X -0.173,Y -348.793,Z 1460.075,A 0.000,B 0.000,C 90.000,E1 229.461} C_DIS
LIN {X -0.097,Y -346.185,Z 1460.062,A 0.000,B 0.000,C 90.000,E1 227.148} C_DIS
LIN {X -0.088,Y -345.065,Z 1460.058,A 0.000,B 0.000,C 90.000,E1 226.377} C_DIS
LIN {X 0.094,Y -338.586,Z 1460.030,A 0.000,B 0.000,C 90.000,E1 221.310} C_DIS
LIN {X 0.094,Y -336.840,Z 1460.019,A 0.000,B 0.000,C 90.000,E1 219.358} C_DIS
LIN {X 0.014,Y -330.861,Z 1459.988,A 0.000,B 0.000,C 90.000,E1 213.865} C_DIS
LIN {X 0.149,Y -329.296,Z 1459.975,A 0.000,B 0.000,C 90.000,E1 211.465} C_DIS
LIN {X -0.154,Y -324.669,Z 1459.942,A 0.000,B 0.000,C 90.000,E1 205.540} C_DIS
LIN {X 0.174,Y -323.837,Z 1459.928,A 0.000,B 0.000,C 90.000,E1 203.078} C_DIS
LIN {X -0.017,Y -321.124,Z 1459.881,A 0.000,B 0.000,C 90.000,E1 194.662} C_DIS
LIN {X 0.138,Y -320.932,Z 1459.877,A 0.000,B 0.000,C 90.000,E1 193.828} C_DIS
LIN {X -0.076,Y -321.562,Z 1459.832,A 0.000,B 0.000,C 90.000,E1 185.796} C_DIS
LIN {X -0.143,Y -324.415,Z 1459.790,A 0.000,B 0.000,C 90.000,E1 178.165} C_DIS
LIN {X -0.141,Y -325.376,Z 1459.783,A 0.000,B 0.000,C 90.000,E1 176.963} C_DIS
LIN {X -0.100,Y -329.112,Z 1459.750,A 0.000,B 0.000,C 90.000,E1 170.971} C_DIS
LIN {X 0.061,Y -334.260,Z 1459.726,A 0.000,B 0.000,C 90.000,E1 166.589} C_DIS
LIN {X 0.067,Y -335.488,Z 1459.719,A 0.000,B 0.000,C 90.000,E1 165.408} C_DIS
LIN {X 0.143,Y -340.932,Z 1459.695,A 0.000,B 0.000,C 90.000,E1 161.094} C_DIS
LIN {X -0.172,Y -342.138,Z 1459.691,A 0.000,B 0.000,C 90.000,E1 160.369} C_DIS
LIN {X -0.056,Y -344.282,Z 1459.681,A 0.000,B 0.000,C 90.000,E1 158.592} C_DIS
LIN {X -0.111,Y -441.885,Z 1459.681,A 0.000,B 0.000,C 90.000,E1 158.592} C_DIS
LIN {X 0.205,Y -445.623,Z 1459.681,A 0.000,B 0.000,C 90.000,E1 158.465} C_DIS
LIN {X -0.058,Y -447.859,Z 1459.680,A 0.000,B 0.000,C 90.000,E1 158.411} C_DIS
LIN {X -0.135,Y -450.689,Z 1459.679,A 0.000,B 0.000,C 90.000,E1 158.284} C_DIS
LIN {X -0.028,Y -453.660,Z 1459.678,A 0.000,B 0.000,C 90.000,E1 158.103} C_DIS
LIN {X -0.101,Y -456.670,Z 1459.677,A 0.000,B 0.000,C 90.000,E1 157.922} C_DIS
LIN {X -0.059,Y -462.713,Z 1459.675,A 0.000,B 0.000,C 90.000,E1 157.486} C_DIS
LIN {X 0.159,Y -468.712,Z 1459.672,A 0.000,B 0.000,C 90.000,E1 156.975} C_DIS
LIN {X -0.030,Y -476.219,Z 1459.669,A 0.000,B 0.000,C 90.000,E1 156.357} C_DIS
LIN {X 0.118,Y -485.060,Z 1459.664,A 0.000,B 0.000,C 90.000,E1 155.561} C_DIS
LIN {X -0.071,Y -492.165,Z 1459.661,A 0.000,B 0.000,C 90.000,E1 154.921} C_DIS
LIN {X -0.273,Y -497.662,Z 1459.658,A 0.000,B 0.000,C 90.000,E1 154.409} C_DIS
LIN {X -0.029,Y -503.041,Z 1459.655,A 0.000,B 0.000,C 90.000,E1 153.819} C_DIS
LIN {X -0.177,Y -508.222,Z 1459.651,A 0.000,B 0.000,C 90.000,E1 153.256} C_DIS
LIN {X -0.040,Y -511.972,Z 1459.649,A 0.000,B 0.000,C 90.000,E1 152.794} C_DIS
LIN {X -0.291,Y -516.418,Z 1459.646,A 0.000,B 0.000,C 90.000,E1 152.231} C_DIS
LIN {X -0.273,Y -520.438,Z 1459.642,A 0.000,B 0.000,C 90.000,E1 151.641} C_DIS
LIN {X -0.223,Y -523.971,Z 1459.639,A 0.000,B 0.000,C 90.000,E1 151.051} C_DIS
LIN {X -0.146,Y -527.253,Z 1459.636,A 0.000,B 0.000,C 90.000,E1 150.461} C_DIS
LIN {X -0.081,Y -531.380,Z 1459.631,A 0.000,B 0.000,C 90.000,E1 149.587} C_DIS
LIN {X 0.200,Y -533.316,Z 1459.629,A 0.000,B 0.000,C 90.000,E1 149.125} C_DIS
LIN {X 0.051,Y -536.634,Z 1459.624,A 0.000,B 0.000,C 90.000,E1 148.280} C_DIS
LIN {X 0.043,Y -538.628,Z 1459.621,A 0.000,B 0.000,C 90.000,E1 147.709} C_DIS
LIN {X 0.230,Y -541.287,Z 1459.616,A 0.000,B 0.000,C 90.000,E1 146.834} C_DIS
LIN {X -0.009,Y -543.761,Z 1459.611,A 0.000,B 0.000,C 90.000,E1 146.008} C_DIS
LIN {X -0.225,Y -546.009,Z 1459.606,A 0.000,B 0.000,C 90.000,E1 145.182} C_DIS
LIN {X -0.102,Y -547.959,Z 1459.602,A 0.000,B 0.000,C 90.000,E1 144.322} C_DIS
LIN {X -0.228,Y -550.226,Z 1459.596,A 0.000,B 0.000,C 90.000,E1 143.210} C_DIS
LIN {X -0.001,Y -552.114,Z 1459.589,A 0.000,B 0.000,C 90.000,E1 142.065} C_DIS
LIN {X -0.247,Y -553.358,Z 1459.585,A 0.000,B 0.000,C 90.000,E1 141.251} C_DIS
LIN {X -0.057,Y -554.728,Z 1459.578,A 0.000,B 0.000,C 90.000,E1 140.114} C_DIS
LIN {X 0.232,Y -556.186,Z 1459.571,A 0.000,B 0.000,C 90.000,E1 138.690} C_DIS
LIN {X 0.123,Y -557.465,Z 1459.563,A 0.000,B 0.000,C 90.000,E1 137.310} C_DIS
LIN {X -0.377,Y -558.616,Z 1459.555,A 0.000,B 0.000,C 90.000,E1 135.972} C_DIS
LIN {X -0.135,Y -559.420,Z 1459.549,A 0.000,B 0.000,C 90.000,E1 134.838} C_DIS
LIN {X 0.117,Y -560.132,Z 1459.543,A 0.000,B 0.000,C 90.000,E1 133.704} C_DIS
LIN {X -0.010,Y -560.624,Z 1459.537,A 0.000,B 0.000,C 90.000,E1 132.609} C_DIS
LIN {X -0.132,Y -560.904,Z 1459.531,A 0.000,B 0.000,C 90.000,E1 131.515} C_DIS
LIN {X 0.259,Y -561.092,Z 1459.523,A 0.000,B 0.000,C 90.000,E1 130.092} C_DIS
LIN {X 0.055,Y -561.200,Z 1459.512,A 0.000,B 0.000,C 90.000,E1 128.177} C_DIS
LIN {X 0.096,Y -561.265,Z 1459.505,A 0.000,B 0.000,C 90.000,E1 126.790} C_DIS
LIN {X -0.203,Y -561.166,Z 1459.497,A 0.000,B 0.000,C 90.000,E1 125.438} C_DIS
LIN {X -0.273,Y -560.713,Z 1459.488,A 0.000,B 0.000,C 90.000,E1 123.785} C_DIS
LIN {X 0.081,Y -560.369,Z 1459.474,A 0.000,B 0.000,C 90.000,E1 121.258} C_DIS
LIN {X 0.318,Y -560.616,Z 1459.460,A 0.000,B 0.000,C 90.000,E1 118.743} C_DIS
LIN {X -0.030,Y -561.080,Z 1459.448,A 0.000,B 0.000,C 90.000,E1 116.565} C_DIS
LIN {X -0.164,Y -561.671,Z 1459.437,A 0.000,B 0.000,C 90.000,E1 114.643} C_DIS
LIN {X -0.024,Y -562.327,Z 1459.426,A 0.000,B 0.000,C 90.000,E1 112.695} C_DIS
LIN {X -0.096,Y -562.854,Z 1459.417,A 0.000,B 0.000,C 90.000,E1 111.046} C_DIS
LIN {X 0.253,Y -563.197,Z 1459.409,A 0.000,B 0.000,C 90.000,E1 109.631} C_DIS
LIN {X -0.122,Y -563.648,Z 1459.402,A 0.000,B 0.000,C 90.000,E1 108.290} C_DIS
LIN {X 0.329,Y -564.239,Z 1459.391,A 0.000,B 0.000,C 90.000,E1 106.315} C_DIS
LIN {X 0.257,Y -565.102,Z 1459.379,A 0.000,B 0.000,C 90.000,E1 104.120} C_DIS
LIN {X -0.009,Y -565.884,Z 1459.371,A 0.000,B 0.000,C 90.000,E1 102.771} C_DIS
LIN {X -0.220,Y -566.362,Z 1459.368,A 0.000,B 0.000,C 90.000,E1 102.243} C_DIS
LIN {X -0.081,Y -566.927,Z 1459.362,A 0.000,B 0.000,C 90.000,E1 101.130} C_DIS
LIN {X 0.061,Y -567.215,Z 1459.356,A 0.000,B 0.000,C 90.000,E1 100.018} C_DIS
LIN {X 0.278,Y -567.415,Z 1459.348,A 0.000,B 0.000,C 90.000,E1 98.624} C_DIS
LIN {X 0.104,Y -569.309,Z 1459.325,A 0.000,B 0.000,C 90.000,E1 94.531} C_DIS
LIN {X 0.187,Y -570.321,Z 1459.318,A 0.000,B 0.000,C 90.000,E1 93.154} C_DIS
LIN {X 0.146,Y -572.034,Z 1459.306,A 0.000,B 0.000,C 90.000,E1 90.974} C_DIS
LIN {X -0.024,Y -573.597,Z 1459.295,A 0.000,B 0.000,C 90.000,E1 89.083} C_DIS
LIN {X 0.283,Y -574.924,Z 1459.286,A 0.000,B 0.000,C 90.000,E1 87.421} C_DIS
LIN {X 0.076,Y -576.329,Z 1459.277,A 0.000,B 0.000,C 90.000,E1 85.812} C_DIS
LIN {X -0.103,Y -577.712,Z 1459.268,A 0.000,B 0.000,C 90.000,E1 84.204} C_DIS
LIN {X 0.228,Y -578.904,Z 1459.260,A 0.000,B 0.000,C 90.000,E1 82.818} C_DIS
LIN {X 0.230,Y -580.403,Z 1459.251,A 0.000,B 0.000,C 90.000,E1 81.197} C_DIS
LIN {X -0.319,Y -581.923,Z 1459.242,A 0.000,B 0.000,C 90.000,E1 79.634} C_DIS
LIN {X -0.057,Y -583.441,Z 1459.233,A 0.000,B 0.000,C 90.000,E1 77.993} C_DIS
LIN {X 0.000,Y -584.652,Z 1459.226,A 0.000,B 0.000,C 90.000,E1 76.645} C_DIS
LIN {X 0.212,Y -585.658,Z 1459.218,A 0.000,B 0.000,C 90.000,E1 75.283} C_DIS
LIN {X 0.118,Y -586.589,Z 1459.209,A 0.000,B 0.000,C 90.000,E1 73.685} C_DIS
LIN {X 0.285,Y -587.273,Z 1459.203,A 0.000,B 0.000,C 90.000,E1 72.598} C_DIS
LIN {X 0.144,Y -587.956,Z 1459.196,A 0.000,B 0.000,C 90.000,E1 71.275} C_DIS
LIN {X 0.205,Y -588.684,Z 1459.189,A 0.000,B 0.000,C 90.000,E1 69.934} C_DIS
LIN {X -0.176,Y -589.753,Z 1459.178,A 0.000,B 0.000,C 90.000,E1 68.103} C_DIS
LIN {X 0.014,Y -590.582,Z 1459.169,A 0.000,B 0.000,C 90.000,E1 66.485} C_DIS
LIN {X -0.072,Y -591.626,Z 1459.161,A 0.000,B 0.000,C 90.000,E1 64.897} C_DIS
LIN {X -0.128,Y -592.757,Z 1459.152,A 0.000,B 0.000,C 90.000,E1 63.307} C_DIS
LIN {X -0.170,Y -595.165,Z 1459.134,A 0.000,B 0.000,C 90.000,E1 60.127} C_DIS
LIN {X -0.245,Y -596.077,Z 1459.128,A 0.000,B 0.000,C 90.000,E1 59.076} C_DIS
LIN {X 0.124,Y -597.493,Z 1459.119,A 0.000,B 0.000,C 90.000,E1 57.454} C_DIS
LIN {X 0.119,Y -598.588,Z 1459.112,A 0.000,B 0.000,C 90.000,E1 56.135} C_DIS
LIN {X -0.103,Y -599.518,Z 1459.106,A 0.000,B 0.000,C 90.000,E1 55.102} C_DIS
LIN {X -0.077,Y -600.503,Z 1459.099,A 0.000,B 0.000,C 90.000,E1 53.783} C_DIS
LIN {X -0.165,Y -601.391,Z 1459.092,A 0.000,B 0.000,C 90.000,E1 52.477} C_DIS
LIN {X -0.234,Y -602.290,Z 1459.084,A 0.000,B 0.000,C 90.000,E1 51.170} C_DIS
LIN {X -0.163,Y -602.915,Z 1459.078,A 0.000,B 0.000,C 90.000,E1 50.114} C_DIS
LIN {X -0.076,Y -603.220,Z 1459.073,A 0.000,B 0.000,C 90.000,E1 49.057} C_DIS
LIN {X -0.149,Y -603.578,Z 1459.062,A 0.000,B 0.000,C 90.000,E1 47.229} C_DIS
LIN {X 0.343,Y -603.743,Z 1459.057,A 0.000,B 0.000,C 90.000,E1 46.134} C_DIS
LIN {X -0.024,Y -603.617,Z 1459.051,A 0.000,B 0.000,C 90.000,E1 45.121} C_DIS
LIN {X -0.393,Y -603.236,Z 1459.045,A 0.000,B 0.000,C 90.000,E1 44.109} C_DIS
LIN {X 0.092,Y -602.569,Z 1459.039,A 0.000,B 0.000,C 90.000,E1 43.014} C_DIS
LIN {X -0.076,Y -602.037,Z 1459.035,A 0.000,B 0.000,C 90.000,E1 42.243} C_DIS
LIN {X 0.179,Y -600.721,Z 1459.027,A 0.000,B 0.000,C 90.000,E1 40.906} C_DIS
LIN {X -0.162,Y -599.497,Z 1459.022,A 0.000,B 0.000,C 90.000,E1 39.886} C_DIS
LIN {X -0.128,Y -597.288,Z 1459.013,A 0.000,B 0.000,C 90.000,E1 38.302} C_DIS
LIN {X -0.035,Y -595.664,Z 1459.007,A 0.000,B 0.000,C 90.000,E1 37.237} C_DIS
LIN {X -0.183,Y -594.243,Z 1459.002,A 0.000,B 0.000,C 90.000,E1 36.457} C_DIS
LIN {X 0.001,Y -592.626,Z 1458.998,A 0.000,B 0.000,C 90.000,E1 35.644} C_DIS
LIN {X -0.312,Y -590.165,Z 1458.992,A 0.000,B 0.000,C 90.000,E1 34.612} C_DIS
LIN {X 0.163,Y -587.345,Z 1458.986,A 0.000,B 0.000,C 90.000,E1 33.499} C_DIS
LIN {X 0.091,Y -584.916,Z 1458.982,A 0.000,B 0.000,C 90.000,E1 32.704} C_DIS
LIN {X -0.355,Y -583.235,Z 1458.979,A 0.000,B 0.000,C 90.000,E1 32.212} C_DIS
LIN {X -0.157,Y -580.302,Z 1458.974,A 0.000,B 0.000,C 90.000,E1 31.386} C_DIS
LIN {X -0.146,Y -578.220,Z 1458.971,A 0.000,B 0.000,C 90.000,E1 30.846} C_DIS
LIN {X 0.192,Y -574.688,Z 1458.967,A 0.000,B 0.000,C 90.000,E1 30.001} C_DIS
LIN {X -0.042,Y -572.757,Z 1458.965,A 0.000,B 0.000,C 90.000,E1 29.617} C_DIS
LIN {X -0.345,Y -567.784,Z 1458.959,A 0.000,B 0.000,C 90.000,E1 28.693} C_DIS
LIN {X -0.025,Y -564.007,Z 1458.955,A 0.000,B 0.000,C 90.000,E1 27.975} C_DIS
LIN {X 0.056,Y -558.223,Z 1458.950,A 0.000,B 0.000,C 90.000,E1 27.001} C_DIS
LIN {X -0.076,Y -552.792,Z 1458.945,A 0.000,B 0.000,C 90.000,E1 26.181} C_DIS
LIN {X 0.211,Y -548.955,Z 1458.942,A 0.000,B 0.000,C 90.000,E1 25.591} C_DIS
LIN {X 0.040,Y -542.689,Z 1458.938,A 0.000,B 0.000,C 90.000,E1 24.771} C_DIS
LIN {X -0.118,Y -537.137,Z 1458.934,A 0.000,B 0.000,C 90.000,E1 24.079} C_DIS
LIN {X 0.166,Y -531.112,Z 1458.930,A 0.000,B 0.000,C 90.000,E1 23.334} C_DIS
LIN {X 0.235,Y -523.640,Z 1458.925,A 0.000,B 0.000,C 90.000,E1 22.461} C_DIS
LIN {X 0.122,Y -514.601,Z 1458.919,A 0.000,B 0.000,C 90.000,E1 21.482} C_DIS
LIN {X -0.072,Y -506.556,Z 1458.915,A 0.000,B 0.000,C 90.000,E1 20.663} C_DIS
LIN {X -0.004,Y -502.352,Z 1458.912,A 0.000,B 0.000,C 90.000,E1 20.248} C_DIS
LIN {X -0.103,Y -499.280,Z 1458.911,A 0.000,B 0.000,C 90.000,E1 19.993} C_DIS
LIN {X -0.130,Y -494.458,Z 1458.909,A 0.000,B 0.000,C 90.000,E1 19.631} C_DIS
LIN {X -0.040,Y -490.987,Z 1458.908,A 0.000,B 0.000,C 90.000,E1 19.396} C_DIS
LIN {X 0.129,Y -487.808,Z 1458.907,A 0.000,B 0.000,C 90.000,E1 19.214} C_DIS
LIN {X 0.179,Y -485.736,Z 1458.906,A 0.000,B 0.000,C 90.000,E1 19.141} C_DIS
LIN {X 0.025,Y -484.642,Z 1458.906,A 0.000,B 0.000,C 90.000,E1 19.141} C_DIS
LIN {X -0.004,Y -375.130,Z 1458.906,A 0.000,B 0.000,C 90.000,E1 19.141} C_DIS
LIN {X 0.012,Y -373.752,Z 1458.898,A 0.000,B 0.000,C 90.000,E1 17.638} C_DIS
LIN {X -0.041,Y -372.849,Z 1458.894,A 0.000,B 0.000,C 90.000,E1 16.913} C_DIS
LIN {X -0.138,Y -367.589,Z 1458.865,A 0.000,B 0.000,C 90.000,E1 11.771} C_DIS
LIN {X -0.054,Y -366.470,Z 1458.855,A 0.000,B 0.000,C 90.000,E1 9.905} C_DIS
LIN {X -0.116,Y -361.776,Z 1458.822,A 0.000,B 0.000,C 90.000,E1 3.955} C_DIS
LIN {X 0.129,Y -360.896,Z 1458.801,A 0.000,B 0.000,C 90.000,E1 0.172} C_DIS
LIN {X -0.053,Y -359.426,Z 1458.770,A 0.000,B 0.000,C 90.000,E1 354.546} C_DIS
LIN {X 0.070,Y -358.890,Z 1458.759,A 0.000,B 0.000,C 90.000,E1 352.648} C_DIS
LIN {X -0.020,Y -359.563,Z 1458.726,A 0.000,B 0.000,C 90.000,E1 346.645} C_DIS
LIN {X 0.001,Y -361.801,Z 1458.684,A 0.000,B 0.000,C 90.000,E1 339.135} C_DIS
LIN {X -0.154,Y -362.053,Z 1458.680,A 0.000,B 0.000,C 90.000,E1 338.411} C_DIS
LIN {X 0.189,Y -365.980,Z 1458.643,A 0.000,B 0.000,C 90.000,E1 331.641} C_DIS
LIN {X 0.029,Y -366.387,Z 1458.639,A 0.000,B 0.000,C 90.000,E1 330.923} C_DIS
LIN {X -0.031,Y -371.355,Z 1458.604,A 0.000,B 0.000,C 90.000,E1 324.642} C_DIS
LIN {X -0.043,Y -371.766,Z 1458.602,A 0.000,B 0.000,C 90.000,E1 324.276} C_DIS
LIN {X 0.013,Y -377.358,Z 1458.567,A 0.000,B 0.000,C 90.000,E1 318.038} C_DIS
LIN {X 0.012,Y -378.235,Z 1458.563,A 0.000,B 0.000,C 90.000,E1 317.310} C_DIS
LIN {X 0.002,Y -383.940,Z 1458.531,A 0.000,B 0.000,C 90.000,E1 311.515} C_DIS
LIN {X 0.088,Y -384.893,Z 1458.527,A 0.000,B 0.000,C 90.000,E1 310.782} C_DIS
LIN {X 0.262,Y -390.610,Z 1458.495,A 0.000,B 0.000,C 90.000,E1 305.025} C_DIS
LIN {X 0.106,Y -391.104,Z 1458.493,A 0.000,B 0.000,C 90.000,E1 304.692} C_DIS
LIN {X 0.022,Y -391.648,Z 1458.489,A 0.000,B 0.000,C 90.000,E1 303.992} C_DIS
LIN {X -0.080,Y -396.825,Z 1458.459,A 0.000,B 0.000,C 90.000,E1 298.693} C_DIS
LIN {X -0.210,Y -397.120,Z 1458.457,A 0.000,B 0.000,C 90.000,E1 298.359} C_DIS
LIN {X -0.055,Y -401.597,Z 1458.426,A 0.000,B 0.000,C 90.000,E1 292.717} C_DIS
LIN {X 0.222,Y -404.659,Z 1458.395,A 0.000,B 0.000,C 90.000,E1 287.094} C_DIS
LIN {X -0.079,Y -404.735,Z 1458.391,A 0.000,B 0.000,C 90.000,E1 286.441} C_DIS
LIN {X 0.214,Y -406.099,Z 1458.364,A 0.000,B 0.000,C 90.000,E1 281.535} C_DIS
LIN {X -0.176,Y -406.094,Z 1458.362,A 0.000,B 0.000,C 90.000,E1 281.243} C_DIS
LIN {X -0.097,Y -405.680,Z 1458.333,A 0.000,B 0.000,C 90.000,E1 276.024} C_DIS
LIN {X -0.165,Y -405.058,Z 1458.328,A 0.000,B 0.000,C 90.000,E1 274.992} C_DIS
LIN {X -0.060,Y -403.497,Z 1458.304,A 0.000,B 0.000,C 90.000,E1 270.802} C_DIS
LIN {X -0.092,Y -403.288,Z 1458.302,A 0.000,B 0.000,C 90.000,E1 270.458} C_DIS
LIN {X 0.091,Y -398.931,Z 1458.271,A 0.000,B 0.000,C 90.000,E1 264.837} C_DIS
LIN {X -0.040,Y -393.108,Z 1458.242,A 0.000,B 0.000,C 90.000,E1 259.567} C_DIS
LIN {X -0.079,Y -392.835,Z 1458.240,A 0.000,B 0.000,C 90.000,E1 259.218} C_DIS
LIN {X 0.034,Y -385.993,Z 1458.212,A 0.000,B 0.000,C 90.000,E1 254.212} C_DIS
LIN {X -0.026,Y -385.267,Z 1458.208,A 0.000,B 0.000,C 90.000,E1 253.504} C_DIS
LIN {X -0.004,Y -384.768,Z 1458.206,A 0.000,B 0.000,C 90.000,E1 253.142} C_DIS
LIN {X 0.221,Y -377.973,Z 1458.182,A 0.000,B 0.000,C 90.000,E1 248.773} C_DIS
LIN {X -0.044,Y -376.233,Z 1458.174,A 0.000,B 0.000,C 90.000,E1 247.358} C_DIS
LIN {X 0.057,Y -374.944,Z 1458.170,A 0.000,B 0.000,C 90.000,E1 246.613} C_DIS
LIN {X -0.208,Y -368.417,Z 1458.148,A 0.000,B 0.000,C 90.000,E1 242.615} C_DIS
LIN {X 0.097,Y -366.047,Z 1458.137,A 0.000,B 0.000,C 90.000,E1 240.717} C_DIS
LIN {X 0.004,Y -359.196,Z 1458.115,A 0.000,B 0.000,C 90.000,E1 236.628} C_DIS
LIN {X 0.021,Y -355.842,Z 1458.100,A 0.000,B 0.000,C 90.000,E1 233.989} C_DIS
LIN {X -0.173,Y -348.793,Z 1458.075,A 0.000,B 0.000,C 90.000,E1 229.461} C_DIS
LIN {X -0.097,Y -346.185,Z 1458.062,A 0.000,B 0.000,C 90.000,E1 227.148} C_DIS
LIN {X -0.088,Y -345.065,Z 1458.058,A 0.000,B 0.000,C 90.000,E1 226.377} C_DIS
LIN {X 0.094,Y -338.586,Z 1458.030,A 0.000,B 0.000,C 90.000,E1 221.310} C_DIS
LIN {X 0.094,Y -336.840,Z 1458.019,A 0.000,B 0.000,C 90.000,E1 219.358} C_DIS
LIN {X 0.014,Y -330.861,Z 1457.988,A 0.000,B 0.000,C 90.000,E1 213.865} C_DIS
LIN {X 0.149,Y -329.296,Z 1457.975,A 0.000,B 0.000,C 90.000,E1 211.465} C_DIS
LIN {X -0.154,Y -324.669,Z 1457.942,A 0.000,B 0.000,C 90.000,E1 205.540} C_DIS
LIN {X 0.174,Y -323.837,Z 1457.928,A 0.000,B 0.000,C 90.000,E1 203.078} C_DIS
LIN {X -0.017,Y -321.124,Z 1457.881,A 0.000,B 0.000,C 90.000,E1 194.662} C_DIS
LIN {X 0.138,Y -320.932,Z 1457.877,A 0.000,B 0.000,C 90.000,E1 193.828} C_DIS
LIN {X -0.076,Y -321.562,Z 1457.832,A 0.000,B 0.000,C 90.000,E1 185.796} C_DIS
LIN {X -0.143,Y -324.415,Z 1457.790,A 0.000,B 0.000,C 90.000,E1 178.165} C_DIS
LIN {X -0.141,Y -325.376,Z 1457.783,A 0.000,B 0.000,C 90.000,E1 176.963} C_DIS
LIN {X -0.100,Y -329.112,Z 1457.750,A 0.000,B 0.000,C 90.000,E1 170.971} C_DIS
LIN {X 0.061,Y -334.260,Z 1457.726,A 0.000,B 0.000,C 90.000,E1 166.589} C_DIS
LIN {X 0.067,Y -335.488,Z 1457.719,A 0.000,B 0.000,C 90.000,E1 165.408} C_DIS
LIN {X 0.143,Y -340.932,Z 1457.695,A 0.000,B 0.000,C 90.000,E1 161.094} C_DIS
LIN {X -0.172,Y -342.138,Z 1457.691,A 0.000,B 0.000,C 90.000,E1 160.369} C_DIS
LIN {X 0.094,Y -343.526,Z 1457.684,A 0.000,B 0.000,C 90.000,E1 159.156} C_DIS
LIN {X 0.095,Y -435.017,Z 1457.684,A 0.000,B 0.000,C 90.000,E1 159.156} C_DIS
LIN {X 0.092,Y -436.774,Z 1457.684,A 0.000,B 0.000,C 90.000,E1 159.135} C_DIS
LIN {X -0.035,Y -439.314,Z 1457.684,A 0.000,B 0.000,C 90.000,E1 159.082} C_DIS
LIN {X -0.015,Y -443.511,Z 1457.683,A 0.000,B 0.000,C 90.000,E1 158.901} C_DIS
LIN {X 0.131,Y -448.623,Z 1457.681,A 0.000,B 0.000,C 90.000,E1 158.592} C_DIS
LIN {X -0.102,Y -454.663,Z 1457.679,A 0.000,B 0.000,C 90.000,E1 158.209} C_DIS
LIN {X 0.008,Y -460.724,Z 1457.676,A 0.000,B 0.000,C 90.000,E1 157.720} C_DIS
LIN {X -0.107,Y -471.353,Z 1457.671,A 0.000,B 0.000,C 90.000,E1 156.847} C_DIS
LIN {X 0.080,Y -480.302,Z 1457.667,A 0.000,B 0.000,C 90.000,E1 156.049} C_DIS
LIN {X -0.060,Y -487.599,Z 1457.663,A 0.000,B 0.000,C 90.000,E1 155.409} C_DIS
LIN {X 0.000,Y -496.153,Z 1457.659,A 0.000,B 0.000,C 90.000,E1 154.588} C_DIS
LIN {X 0.023,Y -502.871,Z 1457.655,A 0.000,B 0.000,C 90.000,E1 153.896} C_DIS
LIN {X -0.071,Y -508.029,Z 1457.652,A 0.000,B 0.000,C 90.000,E1 153.332} C_DIS
LIN {X 0.111,Y -511.767,Z 1457.649,A 0.000,B 0.000,C 90.000,E1 152.871} C_DIS
LIN {X 0.098,Y -516.277,Z 1457.646,A 0.000,B 0.000,C 90.000,E1 152.281} C_DIS
LIN {X -0.126,Y -520.350,Z 1457.643,A 0.000,B 0.000,C 90.000,E1 151.719} C_DIS
LIN {X 0.015,Y -524.750,Z 1457.639,A 0.000,B 0.000,C 90.000,E1 150.973} C_DIS
LIN {X 0.101,Y -527.957,Z 1457.636,A 0.000,B 0.000,C 90.000,E1 150.383} C_DIS
LIN {X 0.059,Y -531.401,Z 1457.632,A 0.000,B 0.000,C 90.000,E1 149.665} C_DIS
LIN {X 0.192,Y -533.907,Z 1457.628,A 0.000,B 0.000,C 90.000,E1 149.076} C_DIS
LIN {X -0.119,Y -536.195,Z 1457.625,A 0.000,B 0.000,C 90.000,E1 148.535} C_DIS
LIN {X 0.039,Y -538.248,Z 1457.622,A 0.000,B 0.000,C 90.000,E1 147.946} C_DIS
LIN {X -0.239,Y -540.957,Z 1457.617,A 0.000,B 0.000,C 90.000,E1 147.120} C_DIS
LIN {X 0.267,Y -543.460,Z 1457.613,A 0.000,B 0.000,C 90.000,E1 146.215} C_DIS
LIN {X 0.050,Y -545.752,Z 1457.608,A 0.000,B 0.000,C 90.000,E1 145.388} C_DIS
LIN {X -0.147,Y -547.796,Z 1457.603,A 0.000,B 0.000,C 90.000,E1 144.562} C_DIS
LIN {X 0.100,Y -550.607,Z 1457.595,A 0.000,B 0.000,C 90.000,E1 143.130} C_DIS
LIN {X -0.098,Y -552.446,Z 1457.589,A 0.000,B 0.000,C 90.000,E1 142.029} C_DIS
LIN {X 0.096,Y -553.650,Z 1457.584,A 0.000,B 0.000,C 90.000,E1 141.170} C_DIS
LIN {X -0.063,Y -554.983,Z 1457.578,A 0.000,B 0.000,C 90.000,E1 140.070} C_DIS
LIN {X -0.197,Y -556.413,Z 1457.570,A 0.000,B 0.000,C 90.000,E1 138.690} C_DIS
LIN {X -0.303,Y -557.654,Z 1457.563,A 0.000,B 0.000,C 90.000,E1 137.310} C_DIS
LIN {X -0.011,Y -558.771,Z 1457.555,A 0.000,B 0.000,C 90.000,E1 135.891} C_DIS
LIN {X 0.234,Y -559.567,Z 1457.549,A 0.000,B 0.000,C 90.000,E1 134.757} C_DIS
LIN {X 0.155,Y -560.330,Z 1457.541,A 0.000,B 0.000,C 90.000,E1 133.380} C_DIS
LIN {X 0.362,Y -560.699,Z 1457.536,A 0.000,B 0.000,C 90.000,E1 132.528} C_DIS
LIN {X -0.218,Y -560.927,Z 1457.532,A 0.000,B 0.000,C 90.000,E1 131.757} C_DIS
LIN {X -0.161,Y -561.116,Z 1457.523,A 0.000,B 0.000,C 90.000,E1 130.092} C_DIS
LIN {X -0.017,Y -561.214,Z 1457.512,A 0.000,B 0.000,C 90.000,E1 128.141} C_DIS
LIN {X 0.128,Y -561.261,Z 1457.504,A 0.000,B 0.000,C 90.000,E1 126.744} C_DIS
LIN {X -0.165,Y -561.141,Z 1457.497,A 0.000,B 0.000,C 90.000,E1 125.391} C_DIS
LIN {X 0.087,Y -560.701,Z 1457.487,A 0.000,B 0.000,C 90.000,E1 123.706} C_DIS
LIN {X 0.142,Y -560.370,Z 1457.474,A 0.000,B 0.000,C 90.000,E1 121.209} C_DIS
LIN {X 0.103,Y -560.543,Z 1457.461,A 0.000,B 0.000,C 90.000,E1 118.999} C_DIS
LIN {X 0.148,Y -560.855,Z 1457.452,A 0.000,B 0.000,C 90.000,E1 117.334} C_DIS
LIN {X 0.213,Y -561.330,Z 1457.443,A 0.000,B 0.000,C 90.000,E1 115.668} C_DIS
LIN {X -0.270,Y -561.778,Z 1457.435,A 0.000,B 0.000,C 90.000,E1 114.335} C_DIS
LIN {X -0.239,Y -562.251,Z 1457.427,A 0.000,B 0.000,C 90.000,E1 112.950} C_DIS
LIN {X 0.099,Y -562.705,Z 1457.420,A 0.000,B 0.000,C 90.000,E1 111.535} C_DIS
LIN {X -0.081,Y -563.108,Z 1457.412,A 0.000,B 0.000,C 90.000,E1 110.174} C_DIS
LIN {X 0.137,Y -563.771,Z 1457.400,A 0.000,B 0.000,C 90.000,E1 107.946} C_DIS
LIN {X 0.066,Y -564.481,Z 1457.389,A 0.000,B 0.000,C 90.000,E1 106.024} C_DIS
LIN {X -0.154,Y -565.475,Z 1457.378,A 0.000,B 0.000,C 90.000,E1 104.120} C_DIS
LIN {X -0.033,Y -566.108,Z 1457.372,A 0.000,B 0.000,C 90.000,E1 103.008} C_DIS
LIN {X -0.068,Y -567.062,Z 1457.368,A 0.000,B 0.000,C 90.000,E1 102.187} C_DIS
LIN {X 0.058,Y -567.578,Z 1457.367,A 0.000,B 0.000,C 90.000,E1 102.007} C_DIS
LIN {X 0.235,Y -567.807,Z 1457.365,A 0.000,B 0.000,C 90.000,E1 101.715} C_DIS
LIN {X 0.213,Y -567.921,Z 1457.361,A 0.000,B 0.000,C 90.000,E1 100.894} C_DIS
LIN {X 0.188,Y -567.946,Z 1457.356,A 0.000,B 0.000,C 90.000,E1 100.074} C_DIS
LIN {X 0.265,Y -568.055,Z 1457.338,A 0.000,B 0.000,C 90.000,E1 96.777} C_DIS
LIN {X 0.074,Y -569.880,Z 1457.321,A 0.000,B 0.000,C 90.000,E1 93.784} C_DIS
LIN {X 0.146,Y -571.790,Z 1457.307,A 0.000,B 0.000,C 90.000,E1 91.318} C_DIS
LIN {X -0.030,Y -573.352,Z 1457.297,A 0.000,B 0.000,C 90.000,E1 89.427} C_DIS
LIN {X -0.156,Y -574.935,Z 1457.286,A 0.000,B 0.000,C 90.000,E1 87.535} C_DIS
LIN {X 0.213,Y -576.344,Z 1457.277,A 0.000,B 0.000,C 90.000,E1 85.869} C_DIS
LIN {X 0.179,Y -577.978,Z 1457.267,A 0.000,B 0.000,C 90.000,E1 83.976} C_DIS
LIN {X -0.065,Y -579.173,Z 1457.259,A 0.000,B 0.000,C 90.000,E1 82.648} C_DIS
LIN {X -0.064,Y -580.714,Z 1457.250,A 0.000,B 0.000,C 90.000,E1 81.027} C_DIS
LIN {X 0.061,Y -582.232,Z 1457.241,A 0.000,B 0.000,C 90.000,E1 79.398} C_DIS
LIN {X 0.096,Y -583.542,Z 1457.234,A 0.000,B 0.000,C 90.000,E1 78.049} C_DIS
LIN {X 0.158,Y -584.755,Z 1457.226,A 0.000,B 0.000,C 90.000,E1 76.700} C_DIS
LIN {X -0.338,Y -585.774,Z 1457.219,A 0.000,B 0.000,C 90.000,E1 75.408} C_DIS
LIN {X 0.212,Y -586.418,Z 1457.213,A 0.000,B 0.000,C 90.000,E1 74.283} C_DIS
LIN {X -0.275,Y -587.374,Z 1457.204,A 0.000,B 0.000,C 90.000,E1 72.725} C_DIS
LIN {X -0.093,Y -587.931,Z 1457.198,A 0.000,B 0.000,C 90.000,E1 71.638} C_DIS
LIN {X 0.192,Y -588.806,Z 1457.189,A 0.000,B 0.000,C 90.000,E1 70.007} C_DIS
LIN {X -0.092,Y -590.002,Z 1457.177,A 0.000,B 0.000,C 90.000,E1 67.901} C_DIS
LIN {X -0.123,Y -590.836,Z 1457.168,A 0.000,B 0.000,C 90.000,E1 66.305} C_DIS
LIN {X -0.207,Y -591.907,Z 1457.159,A 0.000,B 0.000,C 90.000,E1 64.717} C_DIS
LIN {X -0.264,Y -593.051,Z 1457.151,A 0.000,B 0.000,C 90.000,E1 63.127} C_DIS
LIN {X -0.124,Y -595.014,Z 1457.136,A 0.000,B 0.000,C 90.000,E1 60.461} C_DIS
LIN {X 0.011,Y -596.185,Z 1457.129,A 0.000,B 0.000,C 90.000,E1 59.125} C_DIS
LIN {X 0.070,Y -597.583,Z 1457.120,A 0.000,B 0.000,C 90.000,E1 57.533} C_DIS
LIN {X 0.061,Y -598.707,Z 1457.112,A 0.000,B 0.000,C 90.000,E1 56.215} C_DIS
LIN {X -0.161,Y -599.655,Z 1457.107,A 0.000,B 0.000,C 90.000,E1 55.182} C_DIS
LIN {X 0.219,Y -600.692,Z 1457.099,A 0.000,B 0.000,C 90.000,E1 53.829} C_DIS
LIN {X 0.025,Y -601.718,Z 1457.090,A 0.000,B 0.000,C 90.000,E1 52.271} C_DIS
LIN {X -0.259,Y -602.802,Z 1457.082,A 0.000,B 0.000,C 90.000,E1 50.723} C_DIS
LIN {X -0.178,Y -603.321,Z 1457.076,A 0.000,B 0.000,C 90.000,E1 49.666} C_DIS
LIN {X 0.160,Y -603.527,Z 1457.069,A 0.000,B 0.000,C 90.000,E1 48.324} C_DIS
LIN {X -0.163,Y -603.863,Z 1457.060,A 0.000,B 0.000,C 90.000,E1 46.782} C_DIS
LIN {X 0.093,Y -603.962,Z 1457.056,A 0.000,B 0.000,C 90.000,E1 45.972} C_DIS
LIN {X 0.155,Y -603.797,Z 1457.050,A 0.000,B 0.000,C 90.000,E1 44.919} C_DIS
LIN {X 0.214,Y -603.372,Z 1457.044,A 0.000,B 0.000,C 90.000,E1 43.866} C_DIS
LIN {X -0.151,Y -602.702,Z 1457.038,A 0.000,B 0.000,C 90.000,E1 42.852} C_DIS
LIN {X 0.086,Y -602.081,Z 1457.034,A 0.000,B 0.000,C 90.000,E1 42.043} C_DIS
LIN {X -0.066,Y -600.799,Z 1457.026,A 0.000,B 0.000,C 90.000,E1 40.744} C_DIS
LIN {X -0.023,Y -599.489,Z 1457.021,A 0.000,B 0.000,C 90.000,E1 39.688} C_DIS
LIN {X -0.143,Y -597.681,Z 1457.013,A 0.000,B 0.000,C 90.000,E1 38.382} C_DIS
LIN {X -0.043,Y -596.092,Z 1457.007,A 0.000,B 0.000,C 90.000,E1 37.317} C_DIS
LIN {X 0.168,Y -594.718,Z 1457.003,A 0.000,B 0.000,C 90.000,E1 36.503} C_DIS
LIN {X 0.006,Y -593.107,Z 1456.999,A 0.000,B 0.000,C 90.000,E1 35.724} C_DIS
LIN {X 0.038,Y -590.673,Z 1456.993,A 0.000,B 0.000,C 90.000,E1 34.659} C_DIS
LIN {X 0.382,Y -587.161,Z 1456.985,A 0.000,B 0.000,C 90.000,E1 33.293} C_DIS
LIN {X -0.185,Y -584.676,Z 1456.981,A 0.000,B 0.000,C 90.000,E1 32.546} C_DIS
LIN {X 0.029,Y -582.000,Z 1456.976,A 0.000,B 0.000,C 90.000,E1 31.720} C_DIS
LIN {X -0.093,Y -579.043,Z 1456.972,A 0.000,B 0.000,C 90.000,E1 30.924} C_DIS
LIN {X -0.241,Y -575.487,Z 1456.967,A 0.000,B 0.000,C 90.000,E1 30.129} C_DIS
LIN {X 0.232,Y -572.924,Z 1456.964,A 0.000,B 0.000,C 90.000,E1 29.539} C_DIS
LIN {X -0.075,Y -567.988,Z 1456.959,A 0.000,B 0.000,C 90.000,E1 28.615} C_DIS
LIN {X 0.242,Y -564.204,Z 1456.955,A 0.000,B 0.000,C 90.000,E1 27.897} C_DIS
LIN {X 0.165,Y -559.309,Z 1456.951,A 0.000,B 0.000,C 90.000,E1 27.078} C_DIS
LIN {X 0.291,Y -553.960,Z 1456.946,A 0.000,B 0.000,C 90.000,E1 26.232} C_DIS
LIN {X -0.266,Y -549.191,Z 1456.942,A 0.000,B 0.000,C 90.000,E1 25.591} C_DIS
LIN {X -0.242,Y -544.998,Z 1456.939,A 0.000,B 0.000,C 90.000,E1 25.027} C_DIS
LIN {X 0.037,Y -538.489,Z 1456.934,A 0.000,B 0.000,C 90.000,E1 24.155} C_DIS
LIN {X -0.014,Y -533.808,Z 1456.931,A 0.000,B 0.000,C 90.000,E1 23.590} C_DIS
LIN {X -0.062,Y -525.164,Z 1456.926,A 0.000,B 0.000,C 90.000,E1 22.589} C_DIS
LIN {X -0.180,Y -519.947,Z 1456.922,A 0.000,B 0.000,C 90.000,E1 22.025} C_DIS
LIN {X 0.009,Y -512.122,Z 1456.918,A 0.000,B 0.000,C 90.000,E1 21.153} C_DIS
LIN {X -0.177,Y -501.360,Z 1456.911,A 0.000,B 0.000,C 90.000,E1 20.066} C_DIS
LIN {X -0.030,Y -495.399,Z 1456.908,A 0.000,B 0.000,C 90.000,E1 19.504} C_DIS
LIN {X 0.246,Y -490.727,Z 1456.906,A 0.000,B 0.000,C 90.000,E1 19.087} C_DIS
LIN {X -0.241,Y -487.316,Z 1456.905,A 0.000,B 0.000,C 90.000,E1 18.906} C_DIS
LIN {X -0.048,Y -483.498,Z 1456.904,A 0.000,B 0.000,C 90.000,E1 18.671} C_DIS
LIN {X 0.191,Y -480.817,Z 1456.903,A 0.000,B 0.000,C 90.000,E1 18.544} C_DIS
LIN {X -0.032,Y -479.268,Z 1456.903,A 0.000,B 0.000,C 90.000,E1 18.544} C_DIS
LIN {X -0.054,Y -374.541,Z 1456.903,A 0.000,B 0.000,C 90.000,E1 18.544} C_DIS
LIN {X 0.057,Y -373.437,Z 1456.896,A 0.000,B 0.000,C 90.000,E1 17.330} C_DIS
LIN {X -0.010,Y -367.910,Z 1456.868,A 0.000,B 0.000,C 90.000,E1 12.187} C_DIS
LIN {X 0.010,Y -366.506,Z 1456.855,A 0.000,B 0.000,C 90.000,E1 9.962} C_DIS
LIN {X -0.054,Y -361.806,Z 1456.822,A 0.000,B 0.000,C 90.000,E1 4.012} C_DIS
LIN {X -0.169,Y -360.904,Z 1456.802,A 0.000,B 0.000,C 90.000,E1 0.286} C_DIS
LIN {X -0.053,Y -359.426,Z 1456.770,A 0.000,B 0.000,C 90.000,E1 354.546} C_DIS
LIN {X 0.070,Y -358.890,Z 1456.759,A 0.000,B 0.000,C 90.000,E1 352.648} C_DIS
LIN {X -0.020,Y -359.563,Z 1456.726,A 0.000,B 0.000,C 90.000,E1 346.645} C_DIS
LIN {X 0.001,Y -361.801,Z 1456.684,A 0.000,B 0.000,C 90.000,E1 339.135} C_DIS
LIN {X -0.154,Y -362.053,Z 1456.680,A 0.000,B 0.000,C 90.000,E1 338.411} C_DIS
LIN {X 0.189,Y -365.980,Z 1456.643,A 0.000,B 0.000,C 90.000,E1 331.641} C_DIS
LIN {X 0.029,Y -366.387,Z 1456.639,A 0.000,B 0.000,C 90.000,E1 330.923} C_DIS
LIN {X -0.031,Y -371.355,Z 1456.604,A 0.000,B 0.000,C 90.000,E1 324.642} C_DIS
LIN {X -0.043,Y -371.766,Z 1456.602,A 0.000,B 0.000,C 90.000,E1 324.276} C_DIS
LIN {X 0.013,Y -377.358,Z 1456.567,A 0.000,B 0.000,C 90.000,E1 318.038} C_DIS
LIN {X 0.012,Y -378.235,Z 1456.563,A 0.000,B 0.000,C 90.000,E1 317.310} C_DIS
LIN {X 0.002,Y -383.940,Z 1456.531,A 0.000,B 0.000,C 90.000,E1 311.515} C_DIS
LIN {X 0.088,Y -384.893,Z 1456.527,A 0.000,B 0.000,C 90.000,E1 310.782} C_DIS
LIN {X 0.262,Y -390.610,Z 1456.495,A 0.000,B 0.000,C 90.000,E1 305.025} C_DIS
LIN {X 0.106,Y -391.104,Z 1456.493,A 0.000,B 0.000,C 90.000,E1 304.692} C_DIS
LIN {X 0.022,Y -391.648,Z 1456.489,A 0.000,B 0.000,C 90.000,E1 303.992} C_DIS
LIN {X -0.080,Y -396.825,Z 1456.459,A 0.000,B 0.000,C 90.000,E1 298.693} C_DIS
LIN {X -0.210,Y -397.120,Z 1456.457,A 0.000,B 0.000,C 90.000,E1 298.359} C_DIS
LIN {X -0.055,Y -401.597,Z 1456.426,A 0.000,B 0.000,C 90.000,E1 292.717} C_DIS
LIN {X 0.222,Y -404.659,Z 1456.395,A 0.000,B 0.000,C 90.000,E1 287.094} C_DIS
LIN {X -0.079,Y -404.735,Z 1456.391,A 0.000,B 0.000,C 90.000,E1 286.441} C_DIS
LIN {X 0.214,Y -406.099,Z 1456.364,A 0.000,B 0.000,C 90.000,E1 281.535} C_DIS
LIN {X -0.176,Y -406.094,Z 1456.362,A 0.000,B 0.000,C 90.000,E1 281.243} C_DIS
LIN {X -0.097,Y -405.680,Z 1456.333,A 0.000,B 0.000,C 90.000,E1 276.024} C_DIS
LIN {X -0.165,Y -405.058,Z 1456.328,A 0.000,B 0.000,C 90.000,E1 274.992} C_DIS
LIN {X -0.060,Y -403.497,Z 1456.304,A 0.000,B 0.000,C 90.000,E1 270.802} C_DIS
LIN {X -0.092,Y -403.288,Z 1456.302,A 0.000,B 0.000,C 90.000,E1 270.458} C_DIS
LIN {X 0.091,Y -398.931,Z 1456.271,A 0.000,B 0.000,C 90.000,E1 264.837} C_DIS
LIN {X -0.040,Y -393.108,Z 1456.242,A 0.000,B 0.000,C 90.000,E1 259.567} C_DIS
LIN {X -0.079,Y -392.835,Z 1456.240,A 0.000,B 0.000,C 90.000,E1 259.218} C_DIS
LIN {X 0.034,Y -385.993,Z 1456.212,A 0.000,B 0.000,C 90.000,E1 254.212} C_DIS
LIN {X -0.026,Y -385.267,Z 1456.208,A 0.000,B 0.000,C 90.000,E1 253.504} C_DIS
LIN {X -0.004,Y -384.768,Z 1456.206,A 0.000,B 0.000,C 90.000,E1 253.142} C_DIS
LIN {X 0.221,Y -377.973,Z 1456.182,A 0.000,B 0.000,C 90.000,E1 248.773} C_DIS
LIN {X -0.044,Y -376.233,Z 1456.174,A 0.000,B 0.000,C 90.000,E1 247.358} C_DIS
LIN {X 0.057,Y -374.944,Z 1456.170,A 0.000,B 0.000,C 90.000,E1 246.613} C_DIS
LIN {X -0.208,Y -368.417,Z 1456.148,A 0.000,B 0.000,C 90.000,E1 242.615} C_DIS
LIN {X 0.097,Y -366.047,Z 1456.137,A 0.000,B 0.000,C 90.000,E1 240.717} C_DIS
LIN {X 0.004,Y -359.196,Z 1456.115,A 0.000,B 0.000,C 90.000,E1 236.628} C_DIS
LIN {X 0.021,Y -355.842,Z 1456.100,A 0.000,B 0.000,C 90.000,E1 233.989} C_DIS
LIN {X -0.173,Y -348.793,Z 1456.075,A 0.000,B 0.000,C 90.000,E1 229.461} C_DIS
LIN {X -0.097,Y -346.185,Z 1456.062,A 0.000,B 0.000,C 90.000,E1 227.148} C_DIS
LIN {X -0.088,Y -345.065,Z 1456.058,A 0.000,B 0.000,C 90.000,E1 226.377} C_DIS
LIN {X 0.094,Y -338.586,Z 1456.030,A 0.000,B 0.000,C 90.000,E1 221.310} C_DIS
LIN {X 0.094,Y -336.840,Z 1456.019,A 0.000,B 0.000,C 90.000,E1 219.358} C_DIS
LIN {X 0.014,Y -330.861,Z 1455.988,A 0.000,B 0.000,C 90.000,E1 213.865} C_DIS
LIN {X 0.149,Y -329.296,Z 1455.975,A 0.000,B 0.000,C 90.000,E1 211.465} C_DIS
LIN {X -0.154,Y -324.669,Z 1455.942,A 0.000,B 0.000,C 90.000,E1 205.540} C_DIS
LIN {X 0.174,Y -323.837,Z 1455.928,A 0.000,B 0.000,C 90.000,E1 203.078} C_DIS
LIN {X -0.017,Y -321.124,Z 1455.881,A 0.000,B 0.000,C 90.000,E1 194.662} C_DIS
LIN {X 0.138,Y -320.932,Z 1455.877,A 0.000,B 0.000,C 90.000,E1 193.828} C_DIS
LIN {X -0.076,Y -321.562,Z 1455.832,A 0.000,B 0.000,C 90.000,E1 185.796} C_DIS
LIN {X -0.143,Y -324.415,Z 1455.790,A 0.000,B 0.000,C 90.000,E1 178.165} C_DIS
LIN {X -0.141,Y -325.376,Z 1455.783,A 0.000,B 0.000,C 90.000,E1 176.963} C_DIS
LIN {X -0.100,Y -329.112,Z 1455.750,A 0.000,B 0.000,C 90.000,E1 170.971} C_DIS
